	IF NOT FAULT THEN 
		oaksGVL.rOutdoorTempErrorValue0 := PV; // global utetemp som ställs till 0 vid givarfel.
		oaksGVL.rOutdoorTempErrorValue150 := PV;// global utetemp som ställs till 150 vid givarfel.
	ELSE
		oaksGVL.rOutdoorTempErrorValue0 := 0; // global utetemp som ställs till 0 vid givarfel.
		oaksGVL.rOutdoorTempErrorValue150 := 150;// global utetemp som ställs till 150 vid givarfel.
	END_IF
	oaksGVL.rOutdoorTempMean := PV1; // global medel utetemp
	
	oaksGVL.bOutdoorTempSensorError := FAULT; // globalt utegivarfel

METHOD PRIVATE mMean : BOOL // metod för att sköta uträkning av medelvärde
VAR_INPUT
END_VAR
	FB_BA_GetTime01(bEn :=TRUE);	
	stTime := FB_BA_GetTime01.stSysTi;

	IF stTime.wMinute <> wLastMinuteOfChange THEN
		fbMinuteTrig(CLK := TRUE);
	ELSE
		fbMinuteTrig(CLK := FALSE);
	END_IF
	//4320 minuter - 1 = 72 timmar.
	IF fbMinuteTrig.Q THEN
		FOR iCounter:= iAntalMinuterMedel - 1 TO 1 BY -1 DO
			rArrayMean72Hours[iCounter]:=rArrayMean72Hours[iCounter-1];
		END_FOR;
		rArrayMean72Hours[0] := PV;
		wLastMinuteOfChange := stTime.wMinute;
		IF PV6 < 4320 THEN // Räknas upp för att hålla koll på antal insamlade minuter
			PV6 := PV6 +1;
		END_IF
	END_IF 
	
	lrMeanInternal := 0;
	//4320 minuter - 1 = 72 timmar.
	iAntalMinuterForUtrakning := MIN(iAntalMinuterMedel,PV6); // Max begränsar antal minuter som används för beräkning beroende på hur många minuter som finns insamlade
	FOR iCounter:= iAntalMinuterForUtrakning TO 1 BY -1 DO
		lrMeanInternalTemp := lrMeanInternal;
		lrMeanInternal:=rArrayMean72Hours[iCounter-1] + lrMeanInternalTemp;
	END_FOR;
END_METHOD

//utetemp som behåller sitt senaste giltiga värde vid givarfel 
METHOD PROTECTED mPv : REAL
VAR_INPUT
	bKeepLastValidData : BOOL;
END_VAR



	IF M THEN
		mPv := OPM;
	ELSIF FB_BA_AI01Temperatur.bWireBreak AND NOT bKeepLastValidData THEN
		mPv := 150;
	ELSIF FB_BA_AI01Temperatur.bShortCircuit AND NOT bKeepLastValidData THEN
		mPv := -50;
	ELSE
		mPv := LREAL_TO_REAL(FB_BA_TiAvrg01Temperatur.lrOut) + rCal;
	END_IF
END_METHOD

END_FUNCTION_BLOCK

// oaksLibrary/Givare/fbVoltageLuxLightCon
// 0-10V block med inbyggda taggar för ljusintensitet (lux) med möjlighet att handställa PV-värde och inbyggt lux-villkor för utebelysning. 
//Larmar vid givarfel eller vid handställning.
FUNCTION_BLOCK fbVoltageLuxLightCon
VAR_INPUT
	rLuxScaleX1 : REAL; // Ändra om det är 2-10V exempelvis. Max är 0..32767 så 2-10V = 32767 * 0.2 = 6553
	rLuxScaleX2 : REAL := 32767;
	rLuxScaleMin : REAL := 0;
	rLuxScaleMax : REAL := 10000;
	nErrorConf :UINT;//0=ej givarfel vid scalemin/max, 1=givarefel vid scalemax, 2=givarefel vid scalemin och scalemax
END_VAR
VAR_OUTPUT
	{attribute 'OPC.UA.DA' := '1'}
	PV2 AT %M* : REAL;//Ljusintensitet~wp:[unit]lux[format]0[trendoptions]i:300
	{attribute 'OPC.UA.DA' := '1'}
	AL6 AT %M* : BOOL;//Givarfel luxmätning~wp:
	{attribute 'OPC.UA.DA' := '1'}
	PV8 AT %M* : STRING := '';  //Skalning lux-givare~wp:
	{attribute 'OPC.UA.DA' := '1'}
	V AT %M* : BOOL; //Belysningssvillkor utebel.~wp:[trendoptions]i:14400, t:1
END_VAR
VAR
	usiStateLux AT %I*: USINT;
	iDataInLux AT %I*: INT;
	usiCtrlLux AT %Q*: USINT;
	iDataOutLux AT %Q*: INT;
	FB_BA_AI01Lux : FB_BA_AI;
	FB_BA_TiAvrg01Lux : tc2_ba.FB_BA_TiAvrg;
	sTempLux : STRING;
	fbTON : TON ; 
	
	fbTonBelysningsvillkor : TON;
	fbTofBelysningsvillkor : TOF;
END_VAR
VAR_INPUT PERSISTENT 
	{attribute 'OPC.UA.DA' := '1'}
	SP2 AT %M* : REAL := 400;//Gränsvärde start utebelysning.~wp:[unit]lux[format]0
	{attribute 'OPC.UA.DA' := '1'}
	SP3 AT %M*: REAL := 30;//Till & frånslag tidsfördr.~wp:[unit]min[format]0
	rCal : REAL; // Kalibrering
	iLuxMedelvardeSekunder : UDINT := 180;
END_VAR

	sTempLux := CONCAT(REAL_TO_STRING(rLuxScaleMin),' - '); 
	PV8 := CONCAT(sTempLux,REAL_TO_STRING(rLuxScaleMax)); 
	FB_BA_AI01Lux(
	TI_usiState:= usiStateLux, 
	TI_iDataIn:= iDataInLux, 
	eTerminal:= 17, 
	eSensor:= 0, (* 0 = pt1000, *)
	bConfigurate:= , 
	rX01:=rLuxScaleX1 , 
	rX02:=rLuxScaleX2 , 
	rY01:= rLuxScaleMin, 
	rY02:= rLuxScaleMax, 
	rOffset:= , 
	rSmoothingFactor:= , 
	udiDecimalPlace:= , 
	bEnLimitCtrl:= , 
	rHighLimit:= , 
	rLowLimit:=, 
	udiDelayLimitCtrl_sec:= , 
	TO_usiCtrl=> usiCtrlLux, 
	TO_iDataOut=> iDataOutLux, 
	rVal=> , 
	bWireBreak=> , 
	bShortCircuit=> , 
	bHighLimit=> , 
	bLowLimit=> , 
	bErr=> , 
	sErrDescr=> );
	
	FB_BA_TiAvrg01Lux(
	bEn:= TRUE, 
	bEnAvrg := TRUE,
	lrIn:=REAL_TO_LREAL(FB_BA_AI01Lux.rVal), 
	udiIntval:=1, 
	udiNumOfElem:= iLuxMedelvardeSekunder, 
	lrOut=> );
	PV2 := LREAL_TO_REAL(FB_BA_TiAvrg01Lux.lrOut) +rCal;
	
	//Givarfel vid rangemin/max
	IF nErrorConf = 1 THEN 
		fbTON.IN := PV2 >= rLuxScaleMin - 1;
	ELSIF nErrorConf = 2 THEN 
		fbTON.IN := (PV2 >= rLuxScaleMin - 1) OR (PV2 <= rLuxScaleMax + 1);
	ELSE
		fbTON.IN := 0;
	END_IF
	
	fbTON(PT := T#5S);
	AL6 := FB_BA_AI01Lux.bWireBreak OR FB_BA_AI01Lux.bShortCircuit OR fbTON.Q;
	
	// Till och frånslagsfördröjning ute utebelysningsvillkor (V)
	fbTonBelysningsvillkor(IN:=PV2 < SP2, PT:=fRealToMinute(SP3) , Q=> , ET=> );
	fbTofBelysningsvillkor(IN:=fbTonBelysningsvillkor.Q , PT:=fRealToMinute(SP3) , Q=>V , ET=> );

END_FUNCTION_BLOCK

// oaksLibrary/Givare/fbVoltage
//Generellt analog-in block för 0-10V/4-20mA mfl. Funktionsblock har möjlighet att handställa PV-värde. Larmar vid givarfel eller vid handställning.
//Funktionsblock hanterar samtliga modultyper tex. KL3454/64. iBusTermType (17=0-10V, 21=4-20mA). Se typer E_BA_Terminal_KL.
FUNCTION_BLOCK fbVoltage
VAR_INPUT
	rScaleX1 : REAL; // Ändra om det är 2-10V exempelvis. Max är 0..32767 så 2-10V = 32767 * 0.2 = 6553
	rScaleX2 : REAL := 32767;
	rScaleMin : REAL;
	rScaleMax : REAL;

	iBusTermType : E_BA_TERMINAL_KL := 17; //Bus-terminal typ
	{attribute 'OPC.UA.DA' := '1'}
	M AT %M* : BOOL;//Handställning~wp:[trendoptions]i:14400, t:1
	
	nErrorConf :UINT;//0=ej givarfel vid scalemin/max, 1=givarefel vid scalemax, 2=givarefel vid scalemin och scalemax
END_VAR
VAR_OUTPUT
	rOutput : REAL;//Utgång knyts till tagg
	{attribute 'OPC.UA.DA' := '1'}
	FAULT AT %M* : BOOL;//Givarfel~wp:
	{attribute 'OPC.UA.DA' := '1'}
	AL8 AT %M* : BOOL; //Givare handställd~wp:[alarmoptions]p:3
	{attribute 'OPC.UA.DA' := '1'}
	PV8 AT %M* : STRING := '';  //Skalning givare~wp:
END_VAR
VAR
	usiState AT %I*: USINT;
	iDataIn AT %I*: INT;
	usiCtrl AT %Q*: USINT;
	iDataOut AT %Q*: INT;
	FB_BA_AI01 : FB_BA_AI;
	FB_BA_TiAvrg01 : tc2_ba.FB_BA_TiAvrg;
	sTemp : STRING;
	fbTON : TON;
END_VAR
VAR_INPUT PERSISTENT 
	rHandsetValue : REAL; //OPM värde
	rCal : REAL; //Kalibrering
	iMedelvardeSekunder : UDINT := 5;
END_VAR

	sTemp := CONCAT(REAL_TO_STRING(rScaleMin),' - '); 
	PV8 := CONCAT(sTemp,REAL_TO_STRING(rScaleMax)); 
	
	FB_BA_AI01(
	TI_usiState:= usiState, 
	TI_iDataIn:= iDataIn, 
	eTerminal:= iBusTermType, 
	eSensor:= 0, (* 0 = pt1000, *)
	bConfigurate:= , 
	rX01:=rScaleX1 , 
	rX02:=rScaleX2 , 
	rY01:= rScaleMin, 
	rY02:= rScaleMax, 
	rOffset:= , 
	rSmoothingFactor:= , 
	udiDecimalPlace:= , 
	bEnLimitCtrl:= , 
	rHighLimit:= , 
	rLowLimit:=, 
	udiDelayLimitCtrl_sec:= , 
	TO_usiCtrl=> usiCtrl, 
	TO_iDataOut=> iDataOut, 
	rVal=> , 
	bWireBreak=> , 
	bShortCircuit=> , 
	bHighLimit=> , 
	bLowLimit=> , 
	bErr=> , 
	sErrDescr=> );
	
	FB_BA_TiAvrg01(
	bEn:= TRUE, 
	bEnAvrg := TRUE,
	lrIn:=REAL_TO_LREAL(FB_BA_AI01.rVal), 
	udiIntval:=1, 
	udiNumOfElem:= iMedelvardeSekunder, 
	lrOut=> );
	
	
	AL8 := M;
	
	IF M THEN
		rOutput := rHandsetValue;
	ELSE 
		rOutput := LREAL_TO_REAL(FB_BA_TiAvrg01.lrOut) + rCal;
	END_IF
	
	//Givarfel vid rangemin/max
	IF nErrorConf = 1 THEN 
		fbTON.IN := rOutput >= rScaleMax - 1;
	ELSIF nErrorConf = 2 THEN 
		fbTON.IN := (rOutput >= rScaleMax - 1) OR (rOutput <= rScaleMin + 1);
	ELSE
		fbTON.IN := 0;
	END_IF
	
	fbTON(PT := T#5S);
	FAULT := FB_BA_AI01.bWireBreak OR FB_BA_AI01.bShortCircuit OR fbTON.Q;

END_FUNCTION_BLOCK

// oaksLibrary/Givare/fbVoltageBar
// 0-10V block med inbyggda taggar för tryck (kPa) med möjlighet att handställa PV-värde. Larmar vid givarfel eller vid handställning.
FUNCTION_BLOCK fbVoltageBar
VAR_INPUT
	rScaleX1 : REAL; // Ändra om det är 2-10V exempelvis. Max är 0..32767 så 2-10V = 32767 * 0.2 = 6553
	rScaleX2 : REAL := 32767;
	rScaleMin : REAL;
	rScaleMax : REAL;
	{attribute 'OPC.UA.DA' := '1'}
	M AT %M* : BOOL;//Handställning~wp:[trendoptions]i:14400, t:1
	nErrorConf :UINT;//0=ej givarfel vid scalemin/max, 1=givarefel vid scalemax, 2=givarefel vid scalemin och scalemax
END_VAR
VAR_OUTPUT
	{attribute 'OPC.UA.DA' := '1'}
	PV AT %M* : REAL;//Tryck~wp:[unit]Bar[format]0.0[trendoptions]i:300
	{attribute 'OPC.UA.DA' := '1'}
	FAULT AT %M* : BOOL;//Givarfel~wp:
	{attribute 'OPC.UA.DA' := '1'}
	AL8 AT %M* : BOOL; //Givare handställd~wp:[alarmoptions]p:3
	{attribute 'OPC.UA.DA' := '1'}
	PV8 AT %M* : STRING := '';  //Skalning givare~wp:
END_VAR
VAR
	fbAlarm2 : fbAlarm; // Larm handställning
	usiState AT %I*: USINT;
	iDataIn AT %I*: INT;
	usiCtrl AT %Q*: USINT;
	iDataOut AT %Q*: INT;
	FB_BA_AI01 : FB_BA_AI;
	FB_BA_TiAvrg01 : tc2_ba.FB_BA_TiAvrg;
	sTemp : STRING;
	fbTON : TON ; 
END_VAR
VAR_INPUT PERSISTENT
	{attribute 'OPC.UA.DA' := '1'}
	OPM AT %M* : REAL;//Värde handställning~wp:[unit]Bar[format]0.0
	rCal : REAL; // Kalibrering
	iMedelvardeSekunder : UDINT := 5;
END_VAR

	sTemp := CONCAT(REAL_TO_STRING(rScaleMin),' - '); 
	PV8 := CONCAT(sTemp,REAL_TO_STRING(rScaleMax)); 

	FB_BA_AI01(
	TI_usiState:= usiState, 
	TI_iDataIn:= iDataIn, 
	eTerminal:= 17, 
	eSensor:= 0, (* 0 = pt1000, *)
	bConfigurate:= , 
	rX01:=rScaleX1 , 
	rX02:=rScaleX2 , 
	rY01:= rScaleMin, 
	rY02:= rScaleMax, 
	rOffset:= , 
	rSmoothingFactor:= , 
	udiDecimalPlace:= , 
	bEnLimitCtrl:= , 
	rHighLimit:= , 
	rLowLimit:=, 
	udiDelayLimitCtrl_sec:= , 
	TO_usiCtrl=> usiCtrl, 
	TO_iDataOut=> iDataOut, 
	rVal=> , 
	bWireBreak=> , 
	bShortCircuit=> , 
	bHighLimit=> , 
	bLowLimit=> , 
	bErr=> , 
	sErrDescr=> );
	
	FB_BA_TiAvrg01(
	bEn:= TRUE, 
	bEnAvrg := TRUE,
	lrIn:=REAL_TO_LREAL(FB_BA_AI01.rVal), 
	udiIntval:=1, 
	udiNumOfElem:= iMedelvardeSekunder, 
	lrOut=> );
	
	
	//Handställningslarm
	fbAlarm2(bInput:=M , tAlarmDelay:= , bAutoReset:=TRUE , bAlarmOutput=>AL8 );
	
	IF M THEN
		PV := OPM;
	ELSE 
		PV := LREAL_TO_REAL(FB_BA_TiAvrg01.lrOut) +rCal;
	END_IF
	
	//Givarfel vid rangemin/max
	IF nErrorConf = 1 THEN 
		fbTON.IN := PV >= rScaleMax - 1;
	ELSIF nErrorConf = 2 THEN 
		fbTON.IN := (PV >= rScaleMax - 1) OR (PV <= rScaleMin + 1);
	ELSE
		fbTON.IN := 0;
	END_IF
	
	fbTON(PT := T#5S);
	FAULT := FB_BA_AI01.bWireBreak OR FB_BA_AI01.bShortCircuit OR fbTON.Q;

END_FUNCTION_BLOCK

// oaksLibrary/Givare/fbVoltageCo
// 0-10V block med inbyggda taggar för Kolmonoxid (ppm) med möjlighet att handställa PV-värde. Larmar vid givarfel eller vid handställning.
FUNCTION_BLOCK fbVoltageCo
VAR_INPUT
	rScaleX1 : REAL; // Ändra om det är 2-10V exempelvis. Max är 0..32767 så 2-10V = 32767 * 0.2 = 6553
	rScaleX2 : REAL := 32767;
	rScaleMin : REAL;
	rScaleMax : REAL;
	{attribute 'OPC.UA.DA' := '1'}
	M AT %M* : BOOL;//Handställning~wp:[trendoptions]i:14400, t:1
	nErrorConf :UINT;//0=ej givarfel vid scalemin/max, 1=givarefel vid scalemax, 2=givarefel vid scalemin och scalemax
END_VAR
VAR_OUTPUT
	{attribute 'OPC.UA.DA' := '1'}
	PV AT %M* : REAL;//Kolmonoxid~wp:[unit]ppm[format]0[trendoptions]i:300
	{attribute 'OPC.UA.DA' := '1'}
	FAULT AT %M* : BOOL;//Givarfel~wp:
	{attribute 'OPC.UA.DA' := '1'}
	AL8 AT %M* : BOOL; //Givare handställd~wp:[alarmoptions]p:3
	{attribute 'OPC.UA.DA' := '1'}
	PV8 AT %M* : STRING := '';  //Skalning givare~wp:
END_VAR
VAR
	fbAlarm2 : fbAlarm; // Larm handställning
	usiState AT %I*: USINT;
	iDataIn AT %I*: INT;
	usiCtrl AT %Q*: USINT;
	iDataOut AT %Q*: INT;
	FB_BA_AI01 : FB_BA_AI;
	FB_BA_TiAvrg01 : tc2_ba.FB_BA_TiAvrg;
	sTemp : STRING;
	fbTON : TON ; 
END_VAR
VAR_INPUT PERSISTENT 
	{attribute 'OPC.UA.DA' := '1'}
	OPM AT %M* : REAL;//Värde handställning~wp:[unit]ppm[format]0
	rCal : REAL; // Kalibrering
	iMedelvardeSekunder : UDINT := 5;
END_VAR

	sTemp := CONCAT(REAL_TO_STRING(rScaleMin),' - '); 
	PV8 := CONCAT(sTemp,REAL_TO_STRING(rScaleMax)); 

	FB_BA_AI01(
	TI_usiState:= usiState, 
	TI_iDataIn:= iDataIn, 
	eTerminal:= 17, 
	eSensor:= 0, (* 0 = pt1000, *)
	bConfigurate:= , 
	rX01:=rScaleX1 , 
	rX02:=rScaleX2 , 
	rY01:= rScaleMin, 
	rY02:= rScaleMax, 
	rOffset:= , 
	rSmoothingFactor:= , 
	udiDecimalPlace:= , 
	bEnLimitCtrl:= , 
	rHighLimit:= , 
	rLowLimit:=, 
	udiDelayLimitCtrl_sec:= , 
	TO_usiCtrl=> usiCtrl, 
	TO_iDataOut=> iDataOut, 
	rVal=> , 
	bWireBreak=> , 
	bShortCircuit=> , 
	bHighLimit=> , 
	bLowLimit=> , 
	bErr=> , 
	sErrDescr=> );
	
	FB_BA_TiAvrg01(
	bEn:= TRUE, 
	bEnAvrg := TRUE,
	lrIn:=REAL_TO_LREAL(FB_BA_AI01.rVal), 
	udiIntval:=1, 
	udiNumOfElem:= iMedelvardeSekunder, 
	lrOut=> );
	
	
	//Handställningslarm
	fbAlarm2(bInput:=M , tAlarmDelay:= , bAutoReset:=TRUE , bAlarmOutput=>AL8 );
	
	IF M THEN
		PV := OPM;
	ELSE 
		PV := LREAL_TO_REAL(FB_BA_TiAvrg01.lrOut) +rCal;
	END_IF
	
	//Givarfel vid rangemin/max
	IF nErrorConf = 1 THEN 
		fbTON.IN := PV >= rScaleMax - 1;
	ELSIF nErrorConf = 2 THEN 
		fbTON.IN := (PV >= rScaleMax - 1) OR (PV <= rScaleMin + 1);
	ELSE
		fbTON.IN := 0;
	END_IF
	
	fbTON(PT := T#5S);
	FAULT := FB_BA_AI01.bWireBreak OR FB_BA_AI01.bShortCircuit OR fbTON.Q;

END_FUNCTION_BLOCK

// oaksLibrary/Givare/fbVoltageCo2
// 0-10V block med inbyggda taggar för tryck (kPa) med möjlighet att handställa PV-värde. Larmar vid givarfel eller vid handställning.
FUNCTION_BLOCK fbVoltageCo2
VAR_INPUT
	rScaleX1 : REAL; // Ändra om det är 2-10V exempelvis. Max är 0..32767 så 2-10V = 32767 * 0.2 = 6553
	rScaleX2 : REAL := 32767;
	rScaleMin : REAL;
	rScaleMax : REAL;
	{attribute 'OPC.UA.DA' := '1'}
	M AT %M* : BOOL;//Handställning~wp:[trendoptions]i:14400, t:1
	nErrorConf :UINT;//0=ej givarfel vid scalemin/max, 1=givarefel vid scalemax, 2=givarefel vid scalemin och scalemax
END_VAR
VAR_OUTPUT
	{attribute 'OPC.UA.DA' := '1'}
	PV AT %M* : REAL;//Co2-halt~wp:[unit]ppm[format]0[trendoptions]i:300
	{attribute 'OPC.UA.DA' := '1'}
	FAULT AT %M* : BOOL;//Givarfel~wp:
	{attribute 'OPC.UA.DA' := '1'}
	AL8 AT %M* : BOOL; //Givare handställd~wp:[alarmoptions]p:3
	{attribute 'OPC.UA.DA' := '1'}
	PV8 AT %M* : STRING := '';  //Skalning givare~wp:
END_VAR
VAR
	fbAlarm2 : fbAlarm; // Larm handställning
	usiState AT %I*: USINT;
	iDataIn AT %I*: INT;
	usiCtrl AT %Q*: USINT;
	iDataOut AT %Q*: INT;
	FB_BA_AI01 : FB_BA_AI;
	FB_BA_TiAvrg01 : tc2_ba.FB_BA_TiAvrg;
	sTemp : STRING;
	fbTON : TON ; 
END_VAR
VAR_INPUT PERSISTENT
	{attribute 'OPC.UA.DA' := '1'}
	OPM AT %M* : REAL;//Värde handställning~wp:[unit]ppm[format]0
	rCal : REAL; // Kalibrering
	iMedelvardeSekunder : UDINT := 5;
END_VAR

	sTemp := CONCAT(REAL_TO_STRING(rScaleMin),' - '); 
	PV8 := CONCAT(sTemp,REAL_TO_STRING(rScaleMax)); 

	FB_BA_AI01(
	TI_usiState:= usiState, 
	TI_iDataIn:= iDataIn, 
	eTerminal:= 17, 
	eSensor:= 0, (* 0 = pt1000, *)
	bConfigurate:= , 
	rX01:=rScaleX1 , 
	rX02:=rScaleX2 , 
	rY01:= rScaleMin, 
	rY02:= rScaleMax, 
	rOffset:= , 
	rSmoothingFactor:= , 
	udiDecimalPlace:= , 
	bEnLimitCtrl:= , 
	rHighLimit:= , 
	rLowLimit:=, 
	udiDelayLimitCtrl_sec:= , 
	TO_usiCtrl=> usiCtrl, 
	TO_iDataOut=> iDataOut, 
	rVal=> , 
	bWireBreak=> , 
	bShortCircuit=> , 
	bHighLimit=> , 
	bLowLimit=> , 
	bErr=> , 
	sErrDescr=> );
	
	FB_BA_TiAvrg01(
	bEn:= TRUE, 
	bEnAvrg := TRUE,
	lrIn:=REAL_TO_LREAL(FB_BA_AI01.rVal), 
	udiIntval:=1, 
	udiNumOfElem:= iMedelvardeSekunder, 
	lrOut=> );
	
	
	//Handställningslarm
	fbAlarm2(bInput:=M , tAlarmDelay:= , bAutoReset:=TRUE , bAlarmOutput=>AL8 );
	
	IF M THEN
		PV := OPM;
	ELSE 
		PV := LREAL_TO_REAL(FB_BA_TiAvrg01.lrOut) +rCal;
	END_IF
	
	//Givarfel vid rangemin/max
	IF nErrorConf = 1 THEN 
		fbTON.IN := PV >= rScaleMax - 1;
	ELSIF nErrorConf = 2 THEN 
		fbTON.IN := (PV >= rScaleMax - 1) OR (PV <= rScaleMin + 1);
	ELSE
		fbTON.IN := 0;
	END_IF
	
	fbTON(PT := T#5S);
	FAULT := FB_BA_AI01.bWireBreak OR FB_BA_AI01.bShortCircuit OR fbTON.Q;

END_FUNCTION_BLOCK

// oaksLibrary/Givare/fbVoltagekPa
// 0-10V block med inbyggda taggar för tryck (kPa) med möjlighet att handställa PV-värde. Larmar vid givarfel eller vid handställning.
FUNCTION_BLOCK fbVoltagekPa
VAR_INPUT
	rScaleX1 : REAL; // Ändra om det är 2-10V exempelvis. Max är 0..32767 så 2-10V = 32767 * 0.2 = 6553
	rScaleX2 : REAL := 32767;
	rScaleMin : REAL;
	rScaleMax : REAL;
	{attribute 'OPC.UA.DA' := '1'}
	M AT %M* : BOOL;//Handställning~wp:[trendoptions]i:14400, t:1
	nErrorConf :UINT;//0=ej givarfel vid scalemin/max, 1=givarefel vid scalemax, 2=givarefel vid scalemin och scalemax
END_VAR
VAR_OUTPUT
	{attribute 'OPC.UA.DA' := '1'}
	PV AT %M* : REAL;//Tryck~wp:[unit]kPa[format]0[trendoptions]i:300
	{attribute 'OPC.UA.DA' := '1'}
	FAULT AT %M* : BOOL;//Givarfel~wp:
	{attribute 'OPC.UA.DA' := '1'}
	AL8 AT %M* : BOOL; //Givare handställd~wp:[alarmoptions]p:3
	{attribute 'OPC.UA.DA' := '1'}
	PV8 AT %M* : STRING := '';  //Skalning givare~wp:
END_VAR
VAR
	fbAlarm2 : fbAlarm; // Larm handställning
	usiState AT %I*: USINT;
	iDataIn AT %I*: INT;
	usiCtrl AT %Q*: USINT;
	iDataOut AT %Q*: INT;
	FB_BA_AI01 : FB_BA_AI;
	FB_BA_TiAvrg01 : tc2_ba.FB_BA_TiAvrg;
	sTemp : STRING;
	fbTON : TON ; 
END_VAR
VAR_INPUT PERSISTENT
	{attribute 'OPC.UA.DA' := '1'} 
	OPM AT %M* : REAL;//Värde handställning~wp:[unit]kPa[format]0
	rCal : REAL; // Kalibrering
	iMedelvardeSekunder : UDINT := 5;
END_VAR

	sTemp := CONCAT(REAL_TO_STRING(rScaleMin),' - '); 
	PV8 := CONCAT(sTemp,REAL_TO_STRING(rScaleMax)); 

	FB_BA_AI01(
	TI_usiState:= usiState, 
	TI_iDataIn:= iDataIn, 
	eTerminal:= 17, 
	eSensor:= 0, (* 0 = pt1000, *)
	bConfigurate:= , 
	rX01:=rScaleX1 , 
	rX02:=rScaleX2 , 
	rY01:= rScaleMin, 
	rY02:= rScaleMax, 
	rOffset:= , 
	rSmoothingFactor:= , 
	udiDecimalPlace:= , 
	bEnLimitCtrl:= , 
	rHighLimit:= , 
	rLowLimit:=, 
	udiDelayLimitCtrl_sec:= , 
	TO_usiCtrl=> usiCtrl, 
	TO_iDataOut=> iDataOut, 
	rVal=> , 
	bWireBreak=> , 
	bShortCircuit=> , 
	bHighLimit=> , 
	bLowLimit=> , 
	bErr=> , 
	sErrDescr=> );
	
	FB_BA_TiAvrg01(
	bEn:= TRUE, 
	bEnAvrg := TRUE,
	lrIn:=REAL_TO_LREAL(FB_BA_AI01.rVal), 
	udiIntval:=1, 
	udiNumOfElem:= iMedelvardeSekunder, 
	lrOut=> );
	
	
	//Handställningslarm
	fbAlarm2(bInput:=M , tAlarmDelay:= , bAutoReset:=TRUE , bAlarmOutput=>AL8 );
	
	IF M THEN
		PV := OPM;
	ELSE 
		PV := LREAL_TO_REAL(FB_BA_TiAvrg01.lrOut) +rCal;
	END_IF
	
	//Givarfel vid rangemin/max
	IF nErrorConf = 1 THEN 
		fbTON.IN := PV >= rScaleMax - 1;
	ELSIF nErrorConf = 2 THEN 
		fbTON.IN := (PV >= rScaleMax - 1) OR (PV <= rScaleMin + 1);
	ELSE
		fbTON.IN := 0;
	END_IF
	
	fbTON(PT := T#5S);
	FAULT := FB_BA_AI01.bWireBreak OR FB_BA_AI01.bShortCircuit OR fbTON.Q;

END_FUNCTION_BLOCK

// oaksLibrary/Givare/fbVoltageLs
//Oaks AB
//2022-03-11
//0-10V block med inbyggda taggar för flöde (L/s) med möjlighet att handställa PV-värde. Larmar vid givarfel eller vid handställning.
FUNCTION_BLOCK fbVoltageLs
VAR_INPUT
	rScaleX1 : REAL; // Ändra om det är 2-10V exempelvis. Max är 0..32767 så 2-10V = 32767 * 0.2 = 6553
	rScaleX2 : REAL := 32767;
	rScaleMin : REAL;
	rScaleMax : REAL;
	{attribute 'OPC.UA.DA' := '1'}
	M AT %M* : BOOL;//Handställning~wp:[trendoptions]i:14400, t:1
	nErrorConf :UINT;//0=ej givarfel vid scalemin/max, 1=givarefel vid scalemax, 2=givarefel vid scalemin och scalemax
END_VAR
VAR_OUTPUT
	{attribute 'OPC.UA.DA' := '1'}
	PV AT %M* : REAL;//Flöde~wp:[unit]l/s[format]0[trendoptions]i:300
	{attribute 'OPC.UA.DA' := '1'}
	FAULT AT %M* : BOOL;//Givarfel~wp:
	{attribute 'OPC.UA.DA' := '1'}
	AL8 AT %M* : BOOL; //Givare handställd~wp:[alarmoptions]p:3
	{attribute 'OPC.UA.DA' := '1'}
	PV8 AT %M* : STRING := '';  //Skalning givare~wp:
END_VAR
VAR
	fbAlarm2 : fbAlarm; //Larm handställning
	usiState AT %I*: USINT;
	iDataIn AT %I*: INT;
	usiCtrl AT %Q*: USINT;
	iDataOut AT %Q*: INT;
	FB_BA_AI01 : FB_BA_AI;
	FB_BA_TiAvrg01 : tc2_ba.FB_BA_TiAvrg;
	sTemp : STRING;
	fbTON : TON ; 
END_VAR
VAR_INPUT PERSISTENT 
	{attribute 'OPC.UA.DA' := '1'}
	OPM AT %M* : REAL;//Värde handställning~wp:[unit]l/s[format]0
	rCal : REAL; // Kalibrering
	iMedelvardeSekunder : UDINT := 5;
END_VAR

	sTemp := CONCAT(REAL_TO_STRING(rScaleMin),' - '); 
	PV8 := CONCAT(sTemp,REAL_TO_STRING(rScaleMax)); 

	FB_BA_AI01(
	TI_usiState:= usiState, 
	TI_iDataIn:= iDataIn, 
	eTerminal:= 17, 
	eSensor:= 0, (* 0 = pt1000, *)
	bConfigurate:= , 
	rX01:=rScaleX1 , 
	rX02:=rScaleX2 , 
	rY01:= rScaleMin, 
	rY02:= rScaleMax, 
	rOffset:= , 
	rSmoothingFactor:= , 
	udiDecimalPlace:= , 
	bEnLimitCtrl:= , 
	rHighLimit:= , 
	rLowLimit:=, 
	udiDelayLimitCtrl_sec:= , 
	TO_usiCtrl=> usiCtrl, 
	TO_iDataOut=> iDataOut, 
	rVal=> , 
	bWireBreak=> , 
	bShortCircuit=> , 
	bHighLimit=> , 
	bLowLimit=> , 
	bErr=> , 
	sErrDescr=> );
	
	FB_BA_TiAvrg01(
	bEn:= TRUE, 
	bEnAvrg := TRUE,
	lrIn:=REAL_TO_LREAL(FB_BA_AI01.rVal), 
	udiIntval:=1, 
	udiNumOfElem:= iMedelvardeSekunder, 
	lrOut=> );
	
	//Handställningslarm
	fbAlarm2(bInput:=M , tAlarmDelay:= , bAutoReset:=TRUE , bAlarmOutput=>AL8 );
	
	IF M THEN
		PV := OPM;
	ELSE 
		PV := LREAL_TO_REAL(FB_BA_TiAvrg01.lrOut) +rCal;
	END_IF
	
	//Givarfel vid rangemin/max
	IF nErrorConf = 1 THEN 
		fbTON.IN := PV >= rScaleMax - 1;
	ELSIF nErrorConf = 2 THEN 
		fbTON.IN := (PV >= rScaleMax - 1) OR (PV <= rScaleMin + 1);
	ELSE
		fbTON.IN := 0;
	END_IF
	
	fbTON(PT := T#5S);
	FAULT := FB_BA_AI01.bWireBreak OR FB_BA_AI01.bShortCircuit OR fbTON.Q;

END_FUNCTION_BLOCK

// oaksLibrary/Givare/fbVoltageLux
// 0-10V block med inbyggda taggar för ljusintensitet (lux) med möjlighet att handställa PV-värde. Larmar vid givarfel eller vid handställning.
FUNCTION_BLOCK fbVoltageLux
VAR_INPUT
	rScaleX1 : REAL; // Ändra om det är 2-10V exempelvis. Max är 0..32767 så 2-10V = 32767 * 0.2 = 6553
	rScaleX2 : REAL := 32767;
	rScaleMin : REAL;
	rScaleMax : REAL;
	{attribute 'OPC.UA.DA' := '1'}
	M AT %M* : BOOL;//Handställning luxgivare~wp:[trendoptions]i:14400, t:1
	nErrorConf :UINT;//0=ej givarfel vid scalemin/max, 1=givarefel vid scalemax, 2=givarefel vid scalemin och scalemax
END_VAR
VAR_OUTPUT
	{attribute 'OPC.UA.DA' := '1'}
	PV AT %M* : REAL;//Ljusintensitet~wp:[unit]lux[format]0[trendoptions]i:300
	{attribute 'OPC.UA.DA' := '1'}
	FAULT AT %M* : BOOL;//Givarfel~wp:
	{attribute 'OPC.UA.DA' := '1'}
	AL8 AT %M* : BOOL; //Givare handställd~wp:[alarmoptions]p:3
	{attribute 'OPC.UA.DA' := '1'}
	PV8 AT %M* : STRING := '';  //Skalning givare~wp:
END_VAR
VAR
	fbAlarm2 : fbAlarm; // Larm handställning
	usiState AT %I*: USINT;
	iDataIn AT %I*: INT;
	usiCtrl AT %Q*: USINT;
	iDataOut AT %Q*: INT;
	FB_BA_AI01 : FB_BA_AI;
	FB_BA_TiAvrg01 : tc2_ba.FB_BA_TiAvrg;
	sTemp : STRING;
	fbTON : TON ; 
END_VAR
VAR_INPUT PERSISTENT 
	{attribute 'OPC.UA.DA' := '1'}
	OPM AT %M* : REAL;//Värde handställning~wp:[unit]lux[format]0
	rCal : REAL; // Kalibrering
	iMedelvardeSekunder : UDINT := 5;
END_VAR

	sTemp := CONCAT(REAL_TO_STRING(rScaleMin),' - '); 
	PV8 := CONCAT(sTemp,REAL_TO_STRING(rScaleMax)); 
	FB_BA_AI01(
	TI_usiState:= usiState, 
	TI_iDataIn:= iDataIn, 
	eTerminal:= 17, 
	eSensor:= 0, (* 0 = pt1000, *)
	bConfigurate:= , 
	rX01:=rScaleX1 , 
	rX02:=rScaleX2 , 
	rY01:= rScaleMin, 
	rY02:= rScaleMax, 
	rOffset:= , 
	rSmoothingFactor:= , 
	udiDecimalPlace:= , 
	bEnLimitCtrl:= , 
	rHighLimit:= , 
	rLowLimit:=, 
	udiDelayLimitCtrl_sec:= , 
	TO_usiCtrl=> usiCtrl, 
	TO_iDataOut=> iDataOut, 
	rVal=> , 
	bWireBreak=> , 
	bShortCircuit=> , 
	bHighLimit=> , 
	bLowLimit=> , 
	bErr=> , 
	sErrDescr=> );
	
	FB_BA_TiAvrg01(
	bEn:= TRUE, 
	bEnAvrg := TRUE,
	lrIn:=REAL_TO_LREAL(FB_BA_AI01.rVal), 
	udiIntval:=1, 
	udiNumOfElem:= iMedelvardeSekunder, 
	lrOut=> );
	
	
	//Handställningslarm
	fbAlarm2(bInput:=M , tAlarmDelay:= , bAutoReset:=TRUE , bAlarmOutput=>AL8 );
	
	IF M THEN
		PV := OPM;
	ELSE 
		PV := LREAL_TO_REAL(FB_BA_TiAvrg01.lrOut) +rCal;
	END_IF
	
	//Givarfel vid rangemin/max
	IF nErrorConf = 1 THEN 
		fbTON.IN := PV >= rScaleMax - 1;
	ELSIF nErrorConf = 2 THEN 
		fbTON.IN := (PV >= rScaleMax - 1) OR (PV <= rScaleMin + 1);
	ELSE
		fbTON.IN := 0;
	END_IF
	
	fbTON(PT := T#5S);
	FAULT := FB_BA_AI01.bWireBreak OR FB_BA_AI01.bShortCircuit OR fbTON.Q;

END_FUNCTION_BLOCK

// oaksLibrary/Givare/fbVoltageNo2
// 0-10V block med inbyggda taggar för Kvävedioxid (ppm) med möjlighet att handställa PV-värde. Larmar vid givarfel eller vid handställning.
FUNCTION_BLOCK fbVoltageNo2
VAR_INPUT
	rScaleX1 : REAL; // Ändra om det är 2-10V exempelvis. Max är 0..32767 så 2-10V = 32767 * 0.2 = 6553
	rScaleX2 : REAL := 32767;
	rScaleMin : REAL;
	rScaleMax : REAL;
	{attribute 'OPC.UA.DA' := '1'}
	M AT %M* : BOOL;//Handställning~wp:[trendoptions]i:14400, t:1
	nErrorConf :UINT;//0=ej givarfel vid scalemin/max, 1=givarefel vid scalemax, 2=givarefel vid scalemin och scalemax
END_VAR
VAR_OUTPUT
	{attribute 'OPC.UA.DA' := '1'}
	PV AT %M* : REAL;//Kvävedioxid~wp:[unit]ppm[format]0.0[trendoptions]i:300
	{attribute 'OPC.UA.DA' := '1'}
	FAULT AT %M* : BOOL;//Givarfel~wp:
	{attribute 'OPC.UA.DA' := '1'}
	AL8 AT %M* : BOOL; //Givare handställd~wp:[alarmoptions]p:3
	{attribute 'OPC.UA.DA' := '1'}
	PV8 AT %M* : STRING := '';  //Skalning givare~wp:
END_VAR
VAR
	fbAlarm2 : fbAlarm; // Larm handställning
	usiState AT %I*: USINT;
	iDataIn AT %I*: INT;
	usiCtrl AT %Q*: USINT;
	iDataOut AT %Q*: INT;
	FB_BA_AI01 : FB_BA_AI;
	FB_BA_TiAvrg01 : tc2_ba.FB_BA_TiAvrg;
	sTemp : STRING;
	fbTON : TON ; 
END_VAR
VAR_INPUT PERSISTENT 
	{attribute 'OPC.UA.DA' := '1'}
	OPM AT %M* : REAL;//Värde handställning~wp:[unit]ppm[format]0.0
	rCal : REAL; // Kalibrering
	iMedelvardeSekunder : UDINT := 5;
END_VAR

	sTemp := CONCAT(REAL_TO_STRING(rScaleMin),' - '); 
	PV8 := CONCAT(sTemp,REAL_TO_STRING(rScaleMax)); 

	FB_BA_AI01(
	TI_usiState:= usiState, 
	TI_iDataIn:= iDataIn, 
	eTerminal:= 17, 
	eSensor:= 0, (* 0 = pt1000, *)
	bConfigurate:= , 
	rX01:=rScaleX1 , 
	rX02:=rScaleX2 , 
	rY01:= rScaleMin, 
	rY02:= rScaleMax, 
	rOffset:= , 
	rSmoothingFactor:= , 
	udiDecimalPlace:= , 
	bEnLimitCtrl:= , 
	rHighLimit:= , 
	rLowLimit:=, 
	udiDelayLimitCtrl_sec:= , 
	TO_usiCtrl=> usiCtrl, 
	TO_iDataOut=> iDataOut, 
	rVal=> , 
	bWireBreak=> , 
	bShortCircuit=> , 
	bHighLimit=> , 
	bLowLimit=> , 
	bErr=> , 
	sErrDescr=> );
	
	FB_BA_TiAvrg01(
	bEn:= TRUE, 
	bEnAvrg := TRUE,
	lrIn:=REAL_TO_LREAL(FB_BA_AI01.rVal), 
	udiIntval:=1, 
	udiNumOfElem:= iMedelvardeSekunder, 
	lrOut=> );
	
	
	//Handställningslarm
	fbAlarm2(bInput:=M , tAlarmDelay:= , bAutoReset:=TRUE , bAlarmOutput=>AL8 );
	
	IF M THEN
		PV := OPM;
	ELSE 
		PV := LREAL_TO_REAL(FB_BA_TiAvrg01.lrOut) +rCal;
	END_IF
	
	//Givarfel vid rangemin/max
	IF nErrorConf = 1 THEN 
		fbTON.IN := PV >= rScaleMax - 1;
	ELSIF nErrorConf = 2 THEN 
		fbTON.IN := (PV >= rScaleMax - 1) OR (PV <= rScaleMin + 1);
	ELSE
		fbTON.IN := 0;
	END_IF
	
	fbTON(PT := T#5S);
	FAULT := FB_BA_AI01.bWireBreak OR FB_BA_AI01.bShortCircuit OR fbTON.Q;

END_FUNCTION_BLOCK

// oaksLibrary/Givare/fbVoltagePa
// 0-10V block med inbyggda taggar för tryck (Pa) med möjlighet att handställa PV-värde. Larmar vid givarfel eller vid handställning.
FUNCTION_BLOCK fbVoltagePa
VAR_INPUT
	rScaleX1 : REAL; // Ändra om det är 2-10V exempelvis. Max är 0..32767 så 2-10V = 32767 * 0.2 = 6553
	rScaleX2 : REAL := 32767;
	rScaleMin : REAL;
	rScaleMax : REAL;
	{attribute 'OPC.UA.DA' := '1'}
	M AT %M* : BOOL;//Handställning~wp:[trendoptions]i:14400, t:1
	nErrorConf :UINT;//0=inget givarefel vid scalemin/max, 1=givarefel vid scalemax, 2=givarefel vid scalemin och scalemax
END_VAR
VAR_OUTPUT
	{attribute 'OPC.UA.DA' := '1'}
	PV AT %M* : REAL;//Tryck~wp:[unit]Pa[format]0[trendoptions]i:300
	{attribute 'OPC.UA.DA' := '1'}
	FAULT AT %M* : BOOL;//Givarfel~wp:
	{attribute 'OPC.UA.DA' := '1'}
	AL8 AT %M* : BOOL; //Givare handställd~wp:[alarmoptions]p:3
	{attribute 'OPC.UA.DA' := '1'}
	PV8 AT %M* : STRING := '';  //Skalning givare~wp:
END_VAR
VAR
	fbAlarm2 : fbAlarm; // Larm handställning
	usiState AT %I*: USINT;
	iDataIn AT %I*: INT;
	usiCtrl AT %Q*: USINT;
	iDataOut AT %Q*: INT;
	FB_BA_AI01 : FB_BA_AI;
	FB_BA_TiAvrg01 : tc2_ba.FB_BA_TiAvrg;
	sTemp : STRING;
	fbTON : TON ; 
END_VAR
VAR_INPUT PERSISTENT 
	{attribute 'OPC.UA.DA' := '1'}
	OPM AT %M* : REAL;//Värde handställning~wp:[unit]Pa[format]0
	rCal : REAL; // Kalibrering
	iMedelvardeSekunder : UDINT := 5;
END_VAR

	sTemp := CONCAT(REAL_TO_STRING(rScaleMin),' - '); 
	PV8 := CONCAT(sTemp,REAL_TO_STRING(rScaleMax)); 

	FB_BA_AI01(
	TI_usiState:= usiState, 
	TI_iDataIn:= iDataIn, 
	eTerminal:= 17, 
	eSensor:= 0, (* 0 = pt1000, *)
	bConfigurate:= , 
	rX01:=rScaleX1 , 
	rX02:=rScaleX2 , 
	rY01:= rScaleMin, 
	rY02:= rScaleMax, 
	rOffset:= , 
	rSmoothingFactor:= , 
	udiDecimalPlace:= , 
	bEnLimitCtrl:= , 
	rHighLimit:= , 
	rLowLimit:=, 
	udiDelayLimitCtrl_sec:= , 
	TO_usiCtrl=> usiCtrl, 
	TO_iDataOut=> iDataOut, 
	rVal=> , 
	bWireBreak=> , 
	bShortCircuit=> , 
	bHighLimit=> , 
	bLowLimit=> , 
	bErr=> , 
	sErrDescr=> );
	
	FB_BA_TiAvrg01(
	bEn:= TRUE, 
	bEnAvrg := TRUE,
	lrIn:=REAL_TO_LREAL(FB_BA_AI01.rVal), 
	udiIntval:=1, 
	udiNumOfElem:= iMedelvardeSekunder, 
	lrOut=> );
	
	
	//Handställningslarm
	fbAlarm2(bInput:=M , tAlarmDelay:= , bAutoReset:=TRUE , bAlarmOutput=>AL8 );
	
	IF M THEN
		PV := OPM;
	ELSE 
		PV := LREAL_TO_REAL(FB_BA_TiAvrg01.lrOut) +rCal;
	END_IF
	
	//Givarfel vid rangemin/max
	IF nErrorConf = 1 THEN 
		fbTON.IN := PV >= rScaleMax - 1;
	ELSIF nErrorConf = 2 THEN 
		fbTON.IN := (PV >= rScaleMax - 1) OR (PV <= rScaleMin + 1);
	ELSE
		fbTON.IN := 0;
	END_IF
	
	fbTON(PT := T#5S);
	FAULT := FB_BA_AI01.bWireBreak OR FB_BA_AI01.bShortCircuit OR fbTON.Q;

END_FUNCTION_BLOCK

// oaksLibrary/Givare/fbVoltagePaFlowLs
// Extendat fbVoltagePa med inbyggd tagg för uträknat flöde. Knyt ditt uträknade värde in på PV1
FUNCTION_BLOCK fbVoltagePaFlowLs EXTENDS fbVoltagePa
VAR_INPUT
	{attribute 'OPC.UA.DA' := '1'}
	PV1 AT %M* : REAL;//Uträknat flöde~wp:[unit]l/s[format]0[trendoptions]i:300
END_VAR
VAR_OUTPUT
END_VAR
VAR
END_VAR

SUPER^();

END_FUNCTION_BLOCK

// oaksLibrary/Givare/fbVoltageRh
// 0-10V block med inbyggda taggar för temperatur (rH%) med möjlighet att handställa PV-värde. Larmar vid givarfel eller vid handställning.
FUNCTION_BLOCK fbVoltageRh
VAR_INPUT
	rScaleX1 : REAL; // Ändra om det är 2-10V exempelvis. Max är 0..32767 så 2-10V = 32767 * 0.2 = 6553
	rScaleX2 : REAL := 32767;
	rScaleMin : REAL;
	rScaleMax : REAL;
	{attribute 'OPC.UA.DA' := '1'}
	M AT %M* : BOOL;//Handställning~wp:[trendoptions]i:14400, t:1
	nErrorConf :UINT;//0=ej givarfel vid scalemin/max, 1=givarefel vid scalemax, 2=givarefel vid scalemin och scalemax
END_VAR
VAR_OUTPUT
	{attribute 'OPC.UA.DA' := '1'}
	PV AT %M* : REAL;//Fukthalt~wp:[unit]rH%[format]0[trendoptions]i:300
	{attribute 'OPC.UA.DA' := '1'}
	FAULT AT %M* : BOOL;//Givarfel~wp:
	{attribute 'OPC.UA.DA' := '1'}
	AL8 AT %M* : BOOL; //Givare handställd~wp:[alarmoptions]p:3
	{attribute 'OPC.UA.DA' := '1'}
	PV8 AT %M* : STRING := '';  //Skalning givare~wp:
END_VAR
VAR
	fbAlarm2 : fbAlarm; // Larm handställning
	usiState AT %I*: USINT;
	iDataIn AT %I*: INT;
	usiCtrl AT %Q*: USINT;
	iDataOut AT %Q*: INT;
	FB_BA_AI01 : FB_BA_AI;
	FB_BA_TiAvrg01 : tc2_ba.FB_BA_TiAvrg;
	sTemp : STRING;
	fbTON : TON ; 
END_VAR
VAR_INPUT PERSISTENT
	{attribute 'OPC.UA.DA' := '1'}
	OPM AT %M* : REAL;//Värde handställning~wp:[unit]rH%[format]0
	rCal : REAL; // Kalibrering
	iMedelvardeSekunder : UDINT := 5;
END_VAR

sTemp := CONCAT(REAL_TO_STRING(rScaleMin),' - '); 
	PV8 := CONCAT(sTemp,REAL_TO_STRING(rScaleMax)); 

	FB_BA_AI01(
	TI_usiState:= usiState, 
	TI_iDataIn:= iDataIn, 
	eTerminal:= 17, 
	eSensor:= 0, (* 0 = pt1000, *)
	bConfigurate:= , 
	rX01:=rScaleX1 , 
	rX02:=rScaleX2 ,  
	rY01:= rScaleMin, 
	rY02:= rScaleMax, 
	rOffset:= , 
	rSmoothingFactor:= , 
	udiDecimalPlace:= , 
	bEnLimitCtrl:= , 
	rHighLimit:= , 
	rLowLimit:=, 
	udiDelayLimitCtrl_sec:= , 
	TO_usiCtrl=> usiCtrl, 
	TO_iDataOut=> iDataOut, 
	rVal=> , 
	bWireBreak=> , 
	bShortCircuit=> , 
	bHighLimit=> , 
	bLowLimit=> , 
	bErr=> , 
	sErrDescr=> );
	
	FB_BA_TiAvrg01(
	bEn:= TRUE, 
	bEnAvrg := TRUE,
	lrIn:=REAL_TO_LREAL(FB_BA_AI01.rVal), 
	udiIntval:=1, 
	udiNumOfElem:= iMedelvardeSekunder, 
	lrOut=> );
	
	
	//Handställningslarm
	fbAlarm2(bInput:=M , tAlarmDelay:= , bAutoReset:=TRUE , bAlarmOutput=>AL8 );
	
	IF M THEN
		PV := OPM;
	ELSE 
		PV := LREAL_TO_REAL(FB_BA_TiAvrg01.lrOut) +rCal;
	END_IF
	
	//Givarfel vid rangemin/max
	IF nErrorConf = 1 THEN 
		fbTON.IN := PV >= rScaleMax - 1;
	ELSIF nErrorConf = 2 THEN 
		fbTON.IN := (PV >= rScaleMax - 1) OR (PV <= rScaleMin + 1);
	ELSE
		fbTON.IN := 0;
	END_IF
	
	fbTON(PT := T#5S);
	FAULT := FB_BA_AI01.bWireBreak OR FB_BA_AI01.bShortCircuit OR fbTON.Q;

END_FUNCTION_BLOCK

// oaksLibrary/Givare/fbVoltageTemp
// 0-10V block med inbyggda taggar för temperatur (°C) med möjlighet att handställa PV-värde. Larmar vid givarfel eller vid handställning.
FUNCTION_BLOCK fbVoltageTemp
VAR_INPUT
	rScaleX1 : REAL; // Ändra om det är 2-10V exempelvis. Max är 0..32767 så 2-10V = 32767 * 0.2 = 6553
	rScaleX2 : REAL := 32767;
	rScaleMin : REAL;
	rScaleMax : REAL;
	{attribute 'OPC.UA.DA' := '1'}
	M AT %M* : BOOL;//Handställning~wp:[trendoptions]i:14400, t:1
	nErrorConf :UINT;//0=ej givarfel vid scalemin/max, 1=givarefel vid scalemax, 2=givarefel vid scalemin och scalemax
END_VAR
VAR_OUTPUT
	{attribute 'OPC.UA.DA' := '1'}
	PV AT %M* : REAL;//Temperatur~wp:[unit]°C[format]0.0[trendoptions]i:300
	{attribute 'OPC.UA.DA' := '1'}
	FAULT AT %M* : BOOL;//Givarfel~wp:
	{attribute 'OPC.UA.DA' := '1'}
	AL8 AT %M* : BOOL; //Givare handställd~wp:[alarmoptions]p:3
	{attribute 'OPC.UA.DA' := '1'}
	PV8 AT %M* : STRING := '';  //Skalning givare~wp:
END_VAR
VAR
	fbAlarm2 : fbAlarm; // Larm handställning
	usiState AT %I*: USINT;
	iDataIn AT %I*: INT;
	usiCtrl AT %Q*: USINT;
	iDataOut AT %Q*: INT;
	FB_BA_AI01 : FB_BA_AI;
	FB_BA_TiAvrg01 : tc2_ba.FB_BA_TiAvrg;
	sTemp : STRING;
	fbTON : TON ; 
END_VAR
VAR_INPUT PERSISTENT 
	{attribute 'OPC.UA.DA' := '1'}
	OPM AT %M* : REAL;//Värde handställning~wp:[unit]°C[format]0.0
	rCal : REAL; // Kalibrering
	iMedelvardeSekunder : UDINT := 5;
END_VAR

	sTemp := CONCAT(REAL_TO_STRING(rScaleMin),' - '); 
	PV8 := CONCAT(sTemp,REAL_TO_STRING(rScaleMax)); 

	FB_BA_AI01(
	TI_usiState:= usiState, 
	TI_iDataIn:= iDataIn, 
	eTerminal:= 17, 
	eSensor:= 0, (* 0 = pt1000, *)
	bConfigurate:= , 
	rX01:=rScaleX1 , 
	rX02:=rScaleX2 , 
	rY01:= rScaleMin, 
	rY02:= rScaleMax, 
	rOffset:= , 
	rSmoothingFactor:= , 
	udiDecimalPlace:= , 
	bEnLimitCtrl:= , 
	rHighLimit:= , 
	rLowLimit:=, 
	udiDelayLimitCtrl_sec:= , 
	TO_usiCtrl=> usiCtrl, 
	TO_iDataOut=> iDataOut, 
	rVal=> , 
	bWireBreak=> , 
	bShortCircuit=> , 
	bHighLimit=> , 
	bLowLimit=> , 
	bErr=> , 
	sErrDescr=> );
	
	FB_BA_TiAvrg01(
	bEn:= TRUE, 
	bEnAvrg := TRUE,
	lrIn:=REAL_TO_LREAL(FB_BA_AI01.rVal), 
	udiIntval:=1, 
	udiNumOfElem:= iMedelvardeSekunder, 
	lrOut=> );
	
	
	//Handställningslarm
	fbAlarm2(bInput:=M , tAlarmDelay:= , bAutoReset:=TRUE , bAlarmOutput=>AL8 );
	
	IF M THEN
		PV := OPM;
	ELSE 
		PV := LREAL_TO_REAL(FB_BA_TiAvrg01.lrOut) +rCal;
	END_IF
	
	//Givarfel vid rangemin/max
	IF nErrorConf = 1 THEN 
		fbTON.IN := PV >= rScaleMax - 1;
	ELSIF nErrorConf = 2 THEN 
		fbTON.IN := (PV >= rScaleMax - 1) OR (PV <= rScaleMin + 1);
	ELSE
		fbTON.IN := 0;
	END_IF
	
	fbTON(PT := T#5S);
	FAULT := FB_BA_AI01.bWireBreak OR FB_BA_AI01.bShortCircuit OR fbTON.Q;

END_FUNCTION_BLOCK

// oaksLibrary/Givare/fbVoltageTempCo2
// 0-10V block med inbyggda taggar för temperatur (°C) och CO2 (ppm) med möjlighet att handställa PV-värde. Larmar vid givarfel eller vid handställning.
FUNCTION_BLOCK fbVoltageTempCo2
VAR_INPUT
	rScaleX1Temperature : REAL; // Ändra om det är 2-10V exempelvis. Max är 0..32767 så 2-10V = 32767 * 0.2 = 6553
	rScaleX2Temperature : REAL := 32767;
	rScaleMinTemperature : REAL:=0;
	rScaleMaxTemperature : REAL:=50;
	
	rScaleX1Co2 : REAL; // Ändra om det är 2-10V exempelvis. Max är 0..32767 så 2-10V = 32767 * 0.2 = 6553
	rScaleX2Co2 : REAL := 32767;
	rScaleMinCo2 : REAL:=0;
	rScaleMaxCo2 : REAL:=2000;
	
	nErrorConfTemp :UINT;//0=inget givarefel 1=givarefel vid Scalemax 2=givarefel vid Scalemin och Scalemax
	nErrorConfCO2 :UINT;//0=inget givarefel 1=givarefel vid Scalemax 2=givarefel vid Scalemin och Scalemax
END_VAR
VAR_OUTPUT
	
	PV AT %M* : REAL;//Temperatur~wp:[unit]°C[format]0.0[trendoptions]i:300
	{attribute 'OPC.UA.DA' := '1'}
	PV1 AT %M* : REAL;//Co2-halt~wp:[unit]ppm[format]0[trendoptions]i:300
	{attribute 'OPC.UA.DA' := '1'}
	FAULT AT %M* : BOOL;//Givarfel temperatur~wp:
	{attribute 'OPC.UA.DA' := '1'}	
	AL8 AT %M* : BOOL;//Givarfel Co2~wp:
	{attribute 'OPC.UA.DA' := '1'}
	PV8 AT %M* : STRING := '';  //Skalning givare~wp:
END_VAR
VAR
	usiStateTemperature AT %I*: USINT;
	iDataInTemperature AT %I*: INT;
	usiCtrlTemperature AT %Q*: USINT;
	iDataOutTemperature AT %Q*: INT;
	FB_BA_AI_Temperature : FB_BA_AI;
	FB_BA_TiAvrgTemperature : tc2_ba.FB_BA_TiAvrg;
	
	usiStateCo2 AT %I*: USINT;
	iDataInCo2 AT %I*: INT;
	usiCtrlCo2 AT %Q*: USINT;
	iDataOutCo2 AT %Q*: INT;
	FB_BA_AI_Co2 : FB_BA_AI;
	FB_BA_TiAvrgCo2 : tc2_ba.FB_BA_TiAvrg;
	sTemp : STRING;
	fbTON1, fbTON2 : TON ;
END_VAR
VAR_INPUT PERSISTENT 
	rCalTemperature : REAL; // Kalibrering
	rCalCo2 : REAL; // Kalibrering
	iMedelvardeSekunder : UDINT := 5;
END_VAR

	

	sTemp := 'Temperatur: ';
	sTemp := CONCAT(CONCAT('Temperatur: ',REAL_TO_STRING(rScaleMinTemperature)),' - '); 
	sTemp := CONCAT(sTemp,REAL_TO_STRING(rScaleMaxTemperature)); 
	sTemp := CONCAT(sTemp,' , CO2: '); 
	sTemp := CONCAT(sTemp,REAL_TO_STRING(rScaleMinCo2)); 
	sTemp := CONCAT(sTemp, ' - ');  
	PV8 := CONCAT(sTemp,REAL_TO_STRING(rScaleMaxCo2));
(*************************** Temperatur *********************)	
	FB_BA_AI_Temperature(
	TI_usiState:= usiStateTemperature, 
	TI_iDataIn:= iDataInTemperature, 
	eTerminal:= 17, 
	eSensor:= 0, (* 0 = pt1000, *)
	bConfigurate:= , 
	rX01:=rScaleX1Temperature , 
	rX02:= rScaleX2Temperature, 
	rY01:= rScaleMinTemperature, 
	rY02:= rScaleMaxTemperature, 
	rOffset:= , 
	rSmoothingFactor:= , 
	udiDecimalPlace:= , 
	bEnLimitCtrl:= , 
	rHighLimit:= , 
	rLowLimit:=, 
	udiDelayLimitCtrl_sec:= , 
	TO_usiCtrl=> usiCtrlTemperature, 
	TO_iDataOut=> iDataOutTemperature, 
	rVal=> , 
	bWireBreak=> , 
	bShortCircuit=> , 
	bHighLimit=> , 
	bLowLimit=> , 
	bErr=> , 
	sErrDescr=> );
	
	FB_BA_TiAvrgTemperature(
	bEn:= TRUE, 
	bEnAvrg := TRUE,
	lrIn:=REAL_TO_LREAL(FB_BA_AI_Temperature.rVal), 
	udiIntval:=1, 
	udiNumOfElem:= iMedelvardeSekunder, 
	lrOut=> );
	
	PV := LREAL_TO_REAL(FB_BA_TiAvrgTemperature.lrOut) +rCalTemperature;
	
	//Givarfel vid rangemin/max
	IF nErrorConfTemp = 1 THEN 
		fbTON1.IN := PV >= rScaleMaxTemperature - 1;
	ELSIF nErrorConfTemp = 2 THEN 
		fbTON1.IN := (PV >= rScaleMaxTemperature - 1) OR (PV <= rScaleMinTemperature + 1);
	ELSE
		fbTON1.IN := 0;
	END_IF
	
	fbTON1(PT := T#5S); 
	
	FAULT := FB_BA_AI_Temperature.bWireBreak OR FB_BA_AI_Temperature.bShortCircuit OR fbTON1.Q;
(*************************** CO2 *********************)	
	FB_BA_AI_Co2(
	TI_usiState:= usiStateCo2, 
	TI_iDataIn:= iDataInCo2, 
	eTerminal:= 17, 
	eSensor:= 0, (* 0 = pt1000, *)
	bConfigurate:= , 
	rX01:= rScaleX1Co2, 
	rX02:= rScaleX2Co2, 
	rY01:= rScaleMinCo2, 
	rY02:= rScaleMaxCo2, 
	rOffset:= , 
	rSmoothingFactor:= , 
	udiDecimalPlace:= , 
	bEnLimitCtrl:= , 
	rHighLimit:= , 
	rLowLimit:=, 
	udiDelayLimitCtrl_sec:= , 
	TO_usiCtrl=> usiCtrlCo2, 
	TO_iDataOut=> iDataOutCo2, 
	rVal=> , 
	bWireBreak=> , 
	bShortCircuit=> , 
	bHighLimit=> , 
	bLowLimit=> , 
	bErr=> , 
	sErrDescr=> );
	
	FB_BA_TiAvrgCo2(
	bEn:= TRUE, 
	bEnAvrg := TRUE,
	lrIn:=REAL_TO_LREAL(FB_BA_AI_Co2.rVal), 
	udiIntval:=1, 
	udiNumOfElem:= iMedelvardeSekunder, 
	lrOut=> );
	
	PV1 := LREAL_TO_REAL(FB_BA_TiAvrgCo2.lrOut) +rCalCo2;
	
	//Givarfel vid rangemin/max
	IF nErrorConfCO2 = 1 THEN 
		fbTON2.IN := PV >= rScaleMaxCo2 - 1;
	ELSIF nErrorConfCO2 = 2 THEN 
		fbTON2.IN := (PV >= rScaleMaxCo2 - 1) OR (PV <= rScaleMinCo2 + 1);
	ELSE
		fbTON2.IN := 0;
	END_IF
	
	fbTON2(PT := T#5S);
	
	AL8 := FB_BA_AI_Co2.bWireBreak OR FB_BA_AI_Co2.bShortCircuit OR fbTON2.Q;

END_FUNCTION_BLOCK

// oaksLibrary/Givare/fbVoltageTempRh
// 0-10V block med inbyggda taggar för temperatur (°C) och rH (rH%) med möjlighet att handställa PV-värde. Larmar vid givarfel eller vid handställning.
FUNCTION_BLOCK fbVoltageTempRh
VAR_INPUT
	rScaleX1Temperature : REAL; // Ändra om det är 2-10V exempelvis. Max är 0..32767 så 2-10V = 32767 * 0.2 = 6553
	rScaleX2Temperature : REAL := 32767;
	rScaleMinTemperature : REAL:=0;
	rScaleMaxTemperature : REAL:=50;
	
	rScaleX1rH : REAL; // Ändra om det är 2-10V exempelvis. Max är 0..32767 så 2-10V = 32767 * 0.2 = 6553
	rScaleX2rH : REAL := 32767;
	rScaleMinrH : REAL:=0;
	rScaleMaxrH : REAL:=100;
	
	nErrorConfTemp :UINT;//0=inget givarefel 1=givarefel vid Scalemax 2=givarefel vid Scalemin och Scalemax
	nErrorConfrH :UINT;//0=inget givarefel 1=givarefel vid Scalemax 2=givarefel vid Scalemin och Scalemax

END_VAR
VAR_OUTPUT
	{attribute 'OPC.UA.DA' := '1'}
	PV AT %M* : REAL;//Temperatur~wp:[unit]°C[format]0.0[trendoptions]i:300
	{attribute 'OPC.UA.DA' := '1'}
	PV1 AT %M* : REAL;//rH-halt~wp:[unit]rH%[format]0[trendoptions]i:300
	{attribute 'OPC.UA.DA' := '1'}
	FAULT AT %M* : BOOL;//Givarfel temperatur~wp:
	{attribute 'OPC.UA.DA' := '1'}
	AL8 AT %M* : BOOL;//Givarfel rH~wp:
	{attribute 'OPC.UA.DA' := '1'}
	PV8 AT %M* : STRING := '';  //Skalning givare~wp:
END_VAR
VAR
	fbAlarm2 : fbAlarm; // Larm handställning
	usiStateTemperature AT %I*: USINT;
	iDataInTemperature AT %I*: INT;
	usiCtrlTemperature AT %Q*: USINT;
	iDataOutTemperature AT %Q*: INT;
	FB_BA_AI_Temperature : FB_BA_AI;
	FB_BA_TiAvrgTemperature : tc2_ba.FB_BA_TiAvrg;
	
	usiStaterH AT %I*: USINT;
	iDataInrH AT %I*: INT;
	usiCtrlrH AT %Q*: USINT;
	iDataOutrH AT %Q*: INT;
	FB_BA_AI_rH : FB_BA_AI;
	FB_BA_TiAvrgrH : tc2_ba.FB_BA_TiAvrg;
	sTemp : STRING;
	fbTON1, fbTON2 : TON ;
END_VAR
VAR_INPUT PERSISTENT 
	rCalTemperature : REAL; // Kalibrering
	rCalrH : REAL; // Kalibrering
	iMedelvardeSekunder : UDINT := 5;
END_VAR

	

	sTemp := 'Temperatur: ';
	sTemp := CONCAT(CONCAT('Temperatur: ',REAL_TO_STRING(rScaleMinTemperature)),' - '); 
	sTemp := CONCAT(sTemp,REAL_TO_STRING(rScaleMaxTemperature)); 
	sTemp := CONCAT(sTemp,' , rH%: '); 
	sTemp := CONCAT(sTemp,REAL_TO_STRING(rScaleMinrH)); 
	sTemp := CONCAT(sTemp, ' - ');  
	PV8 := CONCAT(sTemp,REAL_TO_STRING(rScaleMaxrH));
(*************************** Temperatur *********************)	
	FB_BA_AI_Temperature(
	TI_usiState:= usiStateTemperature, 
	TI_iDataIn:= iDataInTemperature, 
	eTerminal:= 17, 
	eSensor:= 0, (* 0 = pt1000, *)
	bConfigurate:= , 
	rX01:=rScaleX1Temperature , 
	rX02:= rScaleX2Temperature, 
	rY01:= rScaleMinTemperature, 
	rY02:= rScaleMaxTemperature, 
	rOffset:= , 
	rSmoothingFactor:= , 
	udiDecimalPlace:= , 
	bEnLimitCtrl:= , 
	rHighLimit:= , 
	rLowLimit:=, 
	udiDelayLimitCtrl_sec:= , 
	TO_usiCtrl=> usiCtrlTemperature, 
	TO_iDataOut=> iDataOutTemperature, 
	rVal=> , 
	bWireBreak=> , 
	bShortCircuit=> , 
	bHighLimit=> , 
	bLowLimit=> , 
	bErr=> , 
	sErrDescr=> );
	
	FB_BA_TiAvrgTemperature(
	bEn:= TRUE, 
	bEnAvrg := TRUE,
	lrIn:=REAL_TO_LREAL(FB_BA_AI_Temperature.rVal), 
	udiIntval:=1, 
	udiNumOfElem:= iMedelvardeSekunder, 
	lrOut=> );
	
	PV := LREAL_TO_REAL(FB_BA_TiAvrgTemperature.lrOut) +rCalTemperature;
	
	//Givarfel vid rangemin/max
	IF nErrorConfTemp = 1 THEN 
		fbTON1.IN := PV >= rScaleMaxTemperature - 1;
	ELSIF nErrorConfTemp = 2 THEN 
		fbTON1.IN := (PV >= rScaleMaxTemperature - 1) OR (PV <= rScaleMinTemperature + 1);
	ELSE
		fbTON1.IN := 0;
	END_IF
	
	fbTON1(PT := T#5S); 
	
	FAULT := FB_BA_AI_Temperature.bWireBreak OR FB_BA_AI_Temperature.bShortCircuit OR fbTON1.Q;
(*************************** rH *********************)	
	FB_BA_AI_rH(
	TI_usiState:= usiStaterH, 
	TI_iDataIn:= iDataInrH, 
	eTerminal:= 17, 
	eSensor:= 0, (* 0 = pt1000, *)
	bConfigurate:= , 
	rX01:= rScaleX1rH, 
	rX02:= rScaleX2rH, 
	rY01:= rScaleMinrH, 
	rY02:= rScaleMaxrH, 
	rOffset:= , 
	rSmoothingFactor:= , 
	udiDecimalPlace:= , 
	bEnLimitCtrl:= , 
	rHighLimit:= , 
	rLowLimit:=, 
	udiDelayLimitCtrl_sec:= , 
	TO_usiCtrl=> usiCtrlrH, 
	TO_iDataOut=> iDataOutrH, 
	rVal=> , 
	bWireBreak=> , 
	bShortCircuit=> , 
	bHighLimit=> , 
	bLowLimit=> , 
	bErr=> , 
	sErrDescr=> );
	
	FB_BA_TiAvrgrH(
	bEn:= TRUE, 
	bEnAvrg := TRUE,
	lrIn:=REAL_TO_LREAL(FB_BA_AI_rH.rVal), 
	udiIntval:=1, 
	udiNumOfElem:= iMedelvardeSekunder, 
	lrOut=> );
	
	PV1 := LREAL_TO_REAL(FB_BA_TiAvrgrH.lrOut) +rCalrH;
	
	//Givarfel vid rangemin/max
	IF nErrorConfRh = 1 THEN 
		fbTON2.IN := PV >= rScaleMaxrH - 1;
	ELSIF nErrorConfRh = 2 THEN 
		fbTON2.IN := (PV >= rScaleMaxrH - 1) OR (PV <= rScaleMinrH + 1);
	ELSE
		fbTON2.IN := 0;
	END_IF
	
	fbTON2(PT := T#5S);
	
	AL8 := FB_BA_AI_rH.bWireBreak OR FB_BA_AI_rH.bShortCircuit OR fbTON2.Q;

END_FUNCTION_BLOCK

// oaksLibrary/Hämta värde från Webport/fbOutDoorTempMeanFromScada
//Block för att läsa in utetemperatur från Webport. Larm utgår ifall värdet inte uppdateras på 48 timmar (inställningsbart).
(*
Skriv till PV i detta blocket i ett loopande script för uppdateringsvall på 10 sekunder enligt nedan.

tags["TAGG_ATT_HÄMTA_FRÅN_PV"].ReadValue(Moldeo.WebPortCommon.ReadTypes.PRIORITY); 
var copy = tags["TAGG_ATT_HÄMTA_FRÅN_PV"].Value; 
tags["DETTA_BLOCKETS_TAGG_PV"].WriteValue(copy, true); // Exempelvis AS02_GT31_PV

*)
FUNCTION_BLOCK fbOutDoorTempMeanFromScada
VAR_OUTPUT
	{attribute 'OPC.UA.DA' := '1'}
	PV AT %M* : REAL;//Temperatur~wp:[unit]°C[format]0.0[trendoptions]i:300
	{attribute 'OPC.UA.DA' := '1'}
	FAULT AT %M* : BOOL;//Kommunikationsfel hämtning av utetemperatur från webport~wp:
	{attribute 'OPC.UA.DA' := '1'}
	PV1 AT %M*  : REAL; //Medeltemperatur~wp:[unit]°C[format]0.0[trendoptions]i:300
END_VAR
VAR
	fbDifferenceCheckTemp: fbDifferenceCheck;
	fbAlarmTemp : fbAlarm;	

	bResetMeanTemp : BOOL; //Sätt denna till TRUE för återställning av medelvärdesberäkning.
	lrMeanInternal : LREAL;
	lrMeanInternalTemp : LREAL;
	fbPLC_SystemTime: Tc3_BA.FB_BA_GetTime;
	stTime		: tc2_ba.TIMESTRUCT;

	FB_BA_GetTime01 : tc2_ba.FB_BA_GetTime; 
	FB_BA_ExtTiSt01 : tc2_ba.FB_BA_ExtTiSt;	

	
	
	wMinute : WORD;
	fbMinuteTrig : R_TRIG;
	//iTemp : INT;
	iCounter : UINT := 4319;
	
	iAntalMinuterMedel : UINT;
	iAntalMinuterForUtrakning : UINT; //Maxbegränsar antal minuter som används för beräkning beroende på hur många minuter som finns insamlade
END_VAR
VAR PERSISTENT
	wLastMinuteOfChange : WORD;	
	{attribute 'OPC.UA.DA' := '1'}
	PV7 AT %M* : UINT;  //Antal minuter insamlade för medelvärdesberäkning (max 4320)~wp:[unit]minuter[format]0
	{attribute 'OPC.UA.DA' := '1'}
	OPM AT %M* : REAL;//Värde handställning~wp:[unit]°C[format]0.0
	{attribute 'OPC.UA.DA' := '1'}
	SP1 AT %M* : UINT := 12; //Antal timmar för medelvärdesberäkning (2-72)~wp:[unit]timmar[format]0
	
	rArrayMean72Hours : ARRAY [0..4319] OF REAL;
	tAlarmDelayDifferenceCheck : TIME := T#48H;
END_VAR

	// Kollar så värdet uppdateras från överliggande system
	fbDifferenceCheckTemp(rPv:=PV );
	fbAlarmTemp(bInput:= NOT fbDifferenceCheckTemp.bDifference , tAlarmDelay:=tAlarmDelayDifferenceCheck , bAutoReset:=TRUE , bAlarmOutput=>FAULT);
	
	IF bResetMeanTemp THEN
		bResetMeanTemp := FALSE;
		PV7 := 2;
	END_IF

	IF SP1 > 72 THEN // Medelvärdestid maxbegränsas till 72 timmar.
		SP1 := 72;
	ELSIF SP1 < 2 THEN // Medelvärdestid minbegränsas till 2 timmar.
		SP1 := 2;
	END_IF
	
	IF SP1 <= 72 AND SP1 > 1 THEN
		 iAntalMinuterMedel := SP1 * 60;
	END_IF;

	mMean(); // Metod för att räkna ut medelvärde
	//4320 minuter = 72 timmar.
	IF iAntalMinuterForUtrakning > 2 THEN
		PV1 := LREAL_TO_REAL(lrMeanInternal) / iAntalMinuterForUtrakning; 
	END_IF;
	
	oaksGVL.rOutdoorTemp := PV; //utetemp som behåller sitt senaste giltiga värde vid givarfel 
	
	IF NOT FAULT THEN 
		oaksGVL.rOutdoorTempErrorValue0 := PV; // global utetemp som ställs till 0 vid givarfel.
		oaksGVL.rOutdoorTempErrorValue150 := PV;// global utetemp som ställs till 150 vid givarfel.
	ELSE
		oaksGVL.rOutdoorTempErrorValue0 := 0; // global utetemp som ställs till 0 vid givarfel.
		oaksGVL.rOutdoorTempErrorValue150 := 150;// global utetemp som ställs till 150 vid givarfel.
	END_IF
	oaksGVL.rOutdoorTempMean := PV1; // global medel utetemp
	
	oaksGVL.bOutdoorTempSensorError := FAULT; // globalt utegivarfel

METHOD PRIVATE mMean : BOOL // metod för att sköta uträkning av medelvärde
VAR_INPUT
END_VAR
	FB_BA_GetTime01(bEn :=TRUE);	
	stTime := FB_BA_GetTime01.stSysTi;

	IF stTime.wMinute <> wLastMinuteOfChange THEN
		fbMinuteTrig(CLK := TRUE);
	ELSE
		fbMinuteTrig(CLK := FALSE);
	END_IF
	//4320 minuter - 1 = 72 timmar.
	IF fbMinuteTrig.Q THEN
		FOR iCounter:= iAntalMinuterMedel - 1 TO 1 BY -1 DO
			rArrayMean72Hours[iCounter]:=rArrayMean72Hours[iCounter-1];
		END_FOR;
		rArrayMean72Hours[0] := PV;
		wLastMinuteOfChange := stTime.wMinute;
		IF PV7 < 4320 THEN // Räknas upp för att hålla koll på antal insamlade minuter
			PV7 := PV7 +1;
		END_IF
	END_IF 
	
	lrMeanInternal := 0;
	//4320 minuter - 1 = 72 timmar.
	iAntalMinuterForUtrakning := MIN(iAntalMinuterMedel,PV7); // Max begränsar antal minuter som används för beräkning beroende på hur många minuter som finns insamlade
	FOR iCounter:= iAntalMinuterForUtrakning TO 1 BY -1 DO
		lrMeanInternalTemp := lrMeanInternal;
		lrMeanInternal:=rArrayMean72Hours[iCounter-1] + lrMeanInternalTemp;
	END_FOR;
END_METHOD

END_FUNCTION_BLOCK

// oaksLibrary/Larm/Larm med inbyggd larmtagg/fbFreezeAlarm
//Frysvaktsblock med integrerad handställbar pt1000-givare. Handställning förreglas om insignal underskrider 12 grader eller vid givarfel.
//Minbegränsning returtemperatur vid drift stopp aggregat går ej att ställa under 10°C.
FUNCTION_BLOCK fbFreezeAlarm EXTENDS fbPT1000
VAR_INPUT
	bOperationIndication : BOOL; // Driftindikering för tilluftsfläkt kopplas hit. Används för att avgöra vilket minbegränsningsbörvärde som skall användas.
END_VAR
VAR_OUTPUT
	{attribute 'OPC.UA.DA' := '1'}
	LAL AT %M* : BOOL; //Frysvakt~wp:[alarmoptions]p:1,rst:OAKSGVL_RST=1
	rMinOutput : REAL; // Utsignal minbegränsning returvattenregulator 
END_VAR
VAR
	fbReg01 : Tc3_BA_Common.FB_BA_PIDCtrl;
	rSetpoint : REAL;
	fbFreezeInterlock : fbAlarm;
	//itemp :INT;
	{attribute 'OPC.UA.DA' := '1'}
	PV8 AT %M* : REAL; //Aktuell reglersignal minbegränsningsregulator~wp:[unit]%[format]0[trendoptions]i:300
END_VAR
VAR_INPUT PERSISTENT
	{attribute 'OPC.UA.DA' := '1'}
	ALL AT %M* : REAL := 7; //Larmgräns frysvakt~wp:[unit]°C[format]0.0
	{attribute 'OPC.UA.DA' := '1'}
	SP1 AT %M* : REAL := 12; //Minbegränsning returtemperatur vid drift av aggregat~wp:[unit]°C[format]0.0
	{attribute 'OPC.UA.DA' := '1'}
	SP2 AT %M* : REAL := 15; //Minbegränsning returtemperatur vid drift stopp av aggregat~wp:[unit]°C[format]0.0
END_VAR

	SUPER^();

	//Handställning förreglas om insignal underskrider 12 grader eller vid givarfel
	IF FB_BA_AI01.rVal < 12 OR FAULT THEN
		M := FALSE;
	END_IF
	
	// Minbegränsning av frysvaktsinställning 5 grader
	IF ALL < 5.0 THEN 
		ALL := 5.0;
	END_IF

	
	// Frysvaktslarm om temperatur underskrider inställt värde. 
	fbFreezeInterlock(
	bInput:= PV < ALL OR FAULT, 
	tAlarmDelay:= T#3S , 
	bAutoReset:=FALSE , 
	bAlarmOutput=> LAL);
	
	
	// Minbegränsning av inställningsvärde för returtemperatur vid stopp av aggregat
	IF SP2 < 10.0 THEN 
		SP2 := 10.0;
	END_IF
	// Val av börvärde till minbegränsningsregulator
	IF bOperationIndication THEN
		rSetpoint := SP1;
	ELSE
		rSetpoint := SP2;
	END_IF
	
	fbReg01(
	bEn:=TRUE , 
	rW:=rSetpoint , 
	rX:=PV , 
	udiOpMode:= , 
	bActn:= , 
	rKp:= 20, 
	udiTn_ms:= , 
	udiTv_ms:= , 
	udiTd_ms:= , 
	rYMax:=100 , 
	rYMin:= 0, 
	rNZ:= , 
	udiCycCl:= , 
	bSync:= , 
	rSync:= , 
	rY=> , 
	rE=> , 
	bARW=> );
	
	IF NOT FAULT THEN
		rMinOutput := fbReg01.rY;
	ELSE
		rMinOutput := 100;
	END_IF
	// För visning och trendning i webport
	PV8 := rMinOutput;

END_FUNCTION_BLOCK

// oaksLibrary/Larm/Larm med inbyggd larmtagg/fbFreezeAlarmVoltage
//Frysvaktsblock med integrerad handställbar aktiv givare. Handställning förreglas om insignal underskrider 12 grader eller vid givarfel.
//Minbegränsning returtemperatur vid drift stopp aggregat går ej att ställa under 10°C.
FUNCTION_BLOCK fbFreezeAlarmVoltage EXTENDS fbVoltageTemp
VAR_INPUT
	bOperationIndication : BOOL; // Driftindikering för tilluftsfläkt kopplas hit. Används för att avgöra vilket minbegränsningsbörvärde som skall användas.

END_VAR
VAR_OUTPUT
	{attribute 'OPC.UA.DA' := '1'}
	LAL AT %M* : BOOL; //Frysvakt~wp:[alarmoptions]p:1,rst:OAKSGVL_RST=1
	rMinOutput : REAL; // Utsignal minbegränsning returvattenregulator 
END_VAR
VAR
	fbReg01 : Tc3_BA_Common.FB_BA_PIDCtrl;
	rSetpoint : REAL;
	fbFreezeInterlock : fbAlarm;
	//itemp :INT;
	{attribute 'OPC.UA.DA' := '1'}
	PV7 AT %M* : REAL; //Aktuell reglersignal minbegränsningsregulator~wp:[unit]%[format]0[trendoptions]i:300
END_VAR
VAR_INPUT PERSISTENT
	{attribute 'OPC.UA.DA' := '1'}
	ALL AT %M* : REAL := 7; //Larmgräns frysvakt~wp:[unit]°C[format]0.0
	{attribute 'OPC.UA.DA' := '1'}
	SP1 AT %M* : REAL := 12; //Minbegränsning returtemperatur vid drift av aggregat~wp:[unit]°C[format]0.0
	{attribute 'OPC.UA.DA' := '1'}
	SP2 AT %M* : REAL := 15; //Minbegränsning returtemperatur vid drift stopp av aggregat~wp:[unit]°C[format]0.0
END_VAR

	SUPER^();

	//Handställning förreglas om insignal underskrider 12 grader eller vid givarfel
	IF FB_BA_AI01.rVal < 12 OR FAULT THEN
		M := FALSE;
	END_IF
	
	// Minbegränsning av frysvaktsinställning 5 grader
	IF ALL < 5.0 THEN 
		ALL := 5.0;
	END_IF

	
	// Frysvaktslarm om temperatur underskrider inställt värde. 
	fbFreezeInterlock(
	bInput:= PV < ALL OR FAULT, 
	tAlarmDelay:= T#3S , 
	bAutoReset:=FALSE , 
	bAlarmOutput=> LAL);
	
	
	// Minbegränsning av inställningsvärde för returtemperatur vid stopp av aggregat
	IF SP2 < 10.0 THEN 
		SP2 := 10.0;
	END_IF
	// Val av börvärde till minbegränsningsregulator
	IF bOperationIndication THEN
		rSetpoint := SP1;
	ELSE
		rSetpoint := SP2;
	END_IF
	
	fbReg01(
	bEn:=TRUE , 
	rW:=rSetpoint , 
	rX:=PV , 
	udiOpMode:= , 
	bActn:= , 
	rKp:= 20, 
	udiTn_ms:= , 
	udiTv_ms:= , 
	udiTd_ms:= , 
	rYMax:=100 , 
	rYMin:= 0, 
	rNZ:= , 
	udiCycCl:= , 
	bSync:= , 
	rSync:= , 
	rY=> , 
	rE=> , 
	bARW=> );
	
	IF NOT LAL THEN
		rMinOutput := fbReg01.rY;
	ELSE
		rMinOutput := 100;
	END_IF

	// För visning och trendning i webport
	PV7 := rMinOutput;

END_FUNCTION_BLOCK

// oaksLibrary/Larm/Larm med inbyggd larmtagg/fbFusealarm
FUNCTION_BLOCK fbFusealarm
VAR_INPUT
	{attribute 'OPC.UA.DA' := '1'}
	V3 AT %I* : BOOL; //Larmingång~wp:[trendoptions]i:14400, t:1
	bInvert : BOOL;
	bAutoReset : BOOL := TRUE; // Auto-reset av larm
END_VAR
VAR_OUTPUT
	{attribute 'OPC.UA.DA' := '1'}
	AL AT %M*  : BOOL; //Utlöst automatsäkring~wp:
END_VAR
VAR
	bInternalIndication : BOOL;
	fbAlarm1 : fbAlarm;
END_VAR

	IF NOT bInvert THEN
		bInternalIndication :=  V3;
	ELSE
		bInternalIndication := NOT V3;
	END_IF
		
	
	fbAlarm1(
	bInput:= bInternalIndication, 
	tAlarmDelay:= T#500MS, 
	bAutoReset:= bAutoReset, 
	bAlarmOutput=>AL );

END_FUNCTION_BLOCK

// oaksLibrary/Larm/Larm med inbyggd larmtagg/fbJfb
FUNCTION_BLOCK fbJfb
VAR_INPUT
	{attribute 'OPC.UA.DA' := '1'}
	V3 AT %I* : BOOL; //Larmingång~wp:[trendoptions]i:14400, t:1
	bInvert : BOOL;
	bAutoReset : BOOL := TRUE; // Auto-reset av larm
END_VAR
VAR_OUTPUT
	{attribute 'OPC.UA.DA' := '1'}
	AL AT %M*  : BOOL; //Utlöst jordfelsbrytare~wp:
END_VAR
VAR
	bInternalIndication : BOOL;
	fbAlarm1 : fbAlarm;
END_VAR

	IF NOT bInvert THEN
		bInternalIndication :=  V3;
	ELSE
		bInternalIndication := NOT V3;
	END_IF
		
	
	fbAlarm1(
	bInput:= bInternalIndication, 
	tAlarmDelay:= T#500MS, 
	bAutoReset:= bAutoReset, 
	bAlarmOutput=>AL );

END_FUNCTION_BLOCK

// oaksLibrary/Larm/Larm med inbyggd larmtagg/fbLeakDetector
//OAKS AB
//2021-02-08
//Funktionsblock för beräkning av läckage i tex. kallvattensystem
//Funktionen är aktiv mellan inställt intervall för start-/stopptimme (stopptimme avser den timme då funktion stoppar om tex timme 5 ställs stoppar funktion då timme slår om till 5).
//Om inte 0-flöde uppmäts då funktion är aktiv under enligt inställda värden utgår larm.

FUNCTION_BLOCK fbLeakDetector
VAR_INPUT
	iHour : INT; //Aktuell timme
	rVolume : REAL; //Mätarställning från mätare
END_VAR

VAR_INPUT PERSISTENT
	{attribute 'OPC.UA.DA' := '1'}
	SP1 AT %M* : INT := 3; //Starttimme beräkning~wp:[format]0
	{attribute 'OPC.UA.DA' := '1'}
	SP2 AT %M* : INT := 5; //Stopptimme beräkning~wp:[format]0
	{attribute 'OPC.UA.DA' := '1'}
	AHL AT %M* : INT := 3; //Larmgräns antal dagar med fel~wp:[format]0
	{attribute 'OPC.UA.DA' := '1'}
	AD AT %M* : REAL := 5; //Samplingstid nollförbrukning~wp:[format]0[unit]min
END_VAR

VAR_OUTPUT
	{attribute 'OPC.UA.DA' := '1'}
	PV1 AT %M* : INT; //Antal dagar med fel~wp:[format]0
	{attribute 'OPC.UA.DA' := '1'}
	PV8 AT %M* : REAL; //Aktuell differens~wp:[format]0
	{attribute 'OPC.UA.DA' := '1'}
	V AT %M* : BOOL; //Beräkning aktiv~wp:[trendoptions]i:14400, t:1
	{attribute 'OPC.UA.DA' := '1'}
	AL AT %M* : BOOL; //Läckagelarm~wp:[alarmoptions]P:2
END_VAR
VAR
	rNewValue : REAL := 0;
	rStoredValue : REAL := 0;
	bZeroValueOk : BOOL;
	TON_zero : TON;
	F_TRIG_CalcFinished: F_TRIG;
	fbAlarm_Fault : fbAlarm;
	TON_Sampler: TON;
	bReset : BOOL := FALSE;
END_VAR

//Samplingstid
TON_Sampler(IN:= NOT bReset, PT:= T#5S, Q=> , ET=> );
	
	bReset := FALSE;
	
	//Om värden skiljer sig åt
	IF TON_Sampler.Q THEN
		PV8 := rVolume - rStoredValue;	
		rStoredValue := rVolume;
		bReset := TRUE;
	END_IF;

//Starta beräkning 
IF iHour >= SP1 AND iHour < SP2 THEN
	V := TRUE;
ELSE
	//När beräkning ej är aktiv
	V := FALSE; 
END_IF
	
//Beräkning ingen förbrukning under 5 minuter
TON_zero(IN:= (PV8 = 0) AND V,PT:=REAL_TO_TIME(AD*60000) , Q=> , ET=> );

IF TON_zero.Q THEN
	bZeroValueOk := TRUE;
END_IF

//Räkna upp antal dagar det varit fel
F_TRIG_CalcFinished(CLK:= V, Q=> );

IF F_TRIG_CalcFinished.Q AND NOT bZeroValueOk THEN
	PV1 := PV1 + 1;
	//Återställ att värdet är ok inför nästa dag
	bZeroValueOk := FALSE;
ELSIF F_TRIG_CalcFinished.Q AND bZeroValueOk THEN
	PV1 := 0;
	//Återställ att värdet är ok inför nästa dag
	bZeroValueOk := FALSE;
END_IF

//Alarm då antal dagar uppnåtts
fbAlarm_Fault(bInput:= PV1 >= AHL, tAlarmDelay:= T#5S, bAutoReset:= TRUE, bAlarmOutput=> );
AL := fbAlarm_Fault.bAlarmOutput;

END_FUNCTION_BLOCK

// oaksLibrary/Larm/Larm med inbyggd larmtagg/fbManometerLow
FUNCTION_BLOCK fbManometerLow
VAR_INPUT
	{attribute 'OPC.UA.DA' := '1'}
	V3 AT %I* : BOOL; //Larmingång låglarm~wp:[trendoptions]i:14400, t:1
	bInvertLow : BOOL;
	bAutoReset : BOOL := TRUE; // Auto-reset av larm
END_VAR
VAR_OUTPUT
	{attribute 'OPC.UA.DA' := '1'}
	AL AT %M*  : BOOL; //Lågt tryck~wp:
END_VAR
VAR
	bInternalIndicationLow : BOOL;
	fbAlarm1 : fbAlarm;
END_VAR
VAR_INPUT PERSISTENT
	{attribute 'OPC.UA.DA' := '1'}
	AD AT %M*  : REAL := 30; //Larmfördröjning~wp:[unit]sekunder
END_VAR

	IF NOT bInvertLow THEN
		bInternalIndicationLow :=  V3;
	ELSE
		bInternalIndicationLow := NOT V3;
	END_IF
		
	fbAlarm1(
	bInput:= bInternalIndicationLow, 
	tAlarmDelay:= fRealToSecond(rSecond:=AD ), 
	bAutoReset:= bAutoReset, 
	bAlarmOutput=>AL );

END_FUNCTION_BLOCK

// oaksLibrary/Larm/Larm med inbyggd larmtagg/fbManometerLowHigh
FUNCTION_BLOCK fbManometerLowHigh EXTENDS fbManometerLow
VAR_INPUT
	{attribute 'OPC.UA.DA' := '1'}
	V4 AT %I* : BOOL; //Larmingång höglarm~wp:[trendoptions]i:14400, t:1
	bInvertHigh : BOOL;
END_VAR
VAR_OUTPUT
	{attribute 'OPC.UA.DA' := '1'}
	AL1 AT %M*  : BOOL; //Högt tryck~wp:
END_VAR
VAR
	bInternalIndicationHigh : BOOL;
	fbAlarm2 : fbAlarm;
END_VAR

	SUPER^();
	
	IF NOT bInvertHigh THEN
		bInternalIndicationHigh :=  V4;
	ELSE
		bInternalIndicationHigh := NOT V4;
	END_IF
		
	fbAlarm2(bInput:=bInternalIndicationHigh , 
	tAlarmDelay:=fRealToSecond(rSecond:=AD ) , 
	bAutoReset:= bAutoReset,
	bAlarmOutput=>AL1 );

END_FUNCTION_BLOCK

// oaksLibrary/Larm/Larm med inbyggd larmtagg/fbOvervoltageProtection
FUNCTION_BLOCK fbOvervoltageProtection
VAR_INPUT
	{attribute 'OPC.UA.DA' := '1'}
	V3 AT %I* : BOOL; //Larmingång~wp:[trendoptions]i:14400, t:1
	bInvert : BOOL;
	bAutoReset : BOOL := TRUE; // Auto-reset av larm
END_VAR
VAR_OUTPUT
	{attribute 'OPC.UA.DA' := '1'}
	AL AT %M*  : BOOL; //Utlöst överspänningsskydd~wp:
END_VAR
VAR
	bInternalIndication : BOOL;
	fbAlarm1 : fbAlarm;
END_VAR

	IF NOT bInvert THEN
		bInternalIndication :=  V3;
	ELSE
		bInternalIndication := NOT V3;
	END_IF
		
	
	fbAlarm1(
	bInput:= bInternalIndication, 
	tAlarmDelay:= T#500MS, 
	bAutoReset:= bAutoReset, 
	bAlarmOutput=>AL );

END_FUNCTION_BLOCK

// oaksLibrary/Larm/Larm med inbyggd larmtagg/fbRotationGuard
// Block för rotationsvaktslarm VVX.
FUNCTION_BLOCK fbRotationGuard
VAR_INPUT
	rSetpoint : REAL;//Ingång vvx-utsignal
	{attribute 'OPC.UA.DA' := '1'}
	V3 AT %I* : BOOL; //Ingång rotationsvakt~wp:
	bAutoReset : BOOL := TRUE; // Auto-reset av larm
END_VAR
VAR_OUTPUT
	{attribute 'OPC.UA.DA' := '1'}
	AL AT %M*  : BOOL; //Rotationsvakt värmeväxlare~wp:
END_VAR
VAR
	fbAlarm1 : fbAlarm;
	
	fbTonOn : TON;
	fbTonOff : TON;
END_VAR
VAR PERSISTENT
	{attribute 'OPC.UA.DA' := '1'}
	AD AT %M* : REAL := 5; //Larmfördröjning rotationsvakt~wp:[format]0[unit]min
END_VAR

	fbTonOn(IN:= V3 AND rSetpoint = 100, PT:=fRealToMinute(AD)  , Q=> , ET=> );
	fbTonOff(IN:= NOT V3 AND rSetpoint = 100, PT:=fRealToMinute(AD)  , Q=> , ET=> );

	fbAlarm1(
	bInput:= fbTonOn.Q OR fbTonOff.Q, 
	tAlarmDelay:= T#3S, 
	bAutoReset:= bAutoReset, 
	bAlarmOutput=>AL );

END_FUNCTION_BLOCK

// oaksLibrary/Larm/fbDamperAlarmOneInput
// funktionsblock för spjäll-lägeslarm för spjäll med en indikering. Larmar om bDamperOutput är till och bDamperInput inte är till.
FUNCTION_BLOCK fbDamperAlarmOneInput
VAR_INPUT
	bDamperOutput : BOOL;// hit knyts spjällets utsignal
	bDamperInput : BOOL; // hit knyts spjällets indikering
	tAlarmDelay : TIME := T#180S; // Larmfördröjning
	bAutoReset : BOOL; // Ange om larmet ska vara autoresetande.
END_VAR
VAR_OUTPUT
	bDamperAlarm : BOOL; // Larm utgång spjäll i fel läge
END_VAR
VAR
	fbAlarmDelay : TON;
	fbDamperAlarm : fbAlarm; 
END_VAR

fbAlarmDelay(IN:=bDamperOutput AND NOT bDamperInput  , PT:=tAlarmDelay , Q=> , ET=> );

fbDamperAlarm(bInput:= fbAlarmDelay.Q , tAlarmDelay:=T#0S , bAutoReset:=bAutoReset , bAlarmOutput=>bDamperAlarm );

END_FUNCTION_BLOCK

// oaksLibrary/Larm/fbDevAlarm
// Avvikelselarm 
FUNCTION_BLOCK fbDevAlarm EXTENDS fbAlarm
VAR_INPUT
	bEnable : BOOL; // FALSE = larm blockerat
	rProcessValue : REAL; // Ärvärde
	rSetPoint : REAL; // Larmgräns
	rDevLimit : REAL;
	bBlockHighAlarm : BOOL; // Blockera högtemplarm
	bBlockLowAlarm : BOOL; // Blockera lågtemplarm
END_VAR
VAR_OUTPUT
END_VAR
VAR
		iTemp1: INT;
END_VAR

	SUPER^();

	IF rProcessValue > (rSetPoint + rDevLimit) AND bEnable AND NOT bBlockHighAlarm THEN
		bInput := TRUE;
	ELSIF rProcessValue < (rSetPoint - rDevLimit) AND bEnable AND NOT bBlockLowAlarm THEN
		bInput := TRUE;
	ELSE	
		bInput := FALSE;
	END_IF;

END_FUNCTION_BLOCK

// oaksLibrary/Larm/fbDigitalAlarmIO
// Larmblock för digitala larm. Inbyggda taggar för ingång och fördröjning. 
FUNCTION_BLOCK fbDigitalAlarmIO
VAR_INPUT
	{attribute 'OPC.UA.DA' := '1'}
	V3 AT %I* : BOOL; //Larmingång~wp:[trendoptions]i:14400, t:1
	bInvert : BOOL;
	bAutoReset : BOOL := TRUE; // Auto-reset av larm
	bEnable : BOOL := TRUE; 
END_VAR
VAR_OUTPUT
	bOutput : BOOL;
END_VAR
VAR
	bInternalIndication : BOOL;
	fbAlarm1 : fbAlarm;
END_VAR
VAR_INPUT PERSISTENT
	{attribute 'OPC.UA.DA' := '1'}
	AD AT %M* : REAL := 3; //Larmfördröjning~wp:[unit]sekunder[format]0
END_VAR

	IF NOT bInvert THEN
		bInternalIndication :=  V3;
	ELSE
		bInternalIndication := NOT V3;
	END_IF
		
	
	fbAlarm1(
	bInput:= bInternalIndication AND bEnable, 
	tAlarmDelay:= REAL_TO_TIME(AD*1000), 
	bAutoReset:= bAutoReset, 
	bAlarmOutput=>bOutput );

END_FUNCTION_BLOCK

// oaksLibrary/Larm/fbFloorheatHighTemp
//Oaks AB
//2021-09-06
//Funktionsblock för blockering av golvvärme vid hög framledningstemperatur. Då temperatur överstiger inställt värde under 5min blockeras pump i 15 min, funktionen återstartar efter 15min. 
FUNCTION_BLOCK fbFloorheatHighTemp
VAR_INPUT
	rProcessValue : REAL := 3; //Golvvärmetemperatur
	rHighLimit : REAL := 45; //Stopp temperatur
	rLowLimit : REAL := 40; //Start temperatur
END_VAR
VAR_OUTPUT
	bPumpStart : BOOL; //Pumpblockering (True då förregling ej är aktiv)
	PV1 AT %M* : STRING := ' '; //Driftinformation~wp:
	PV8 AT %M* : STRING := ' '; //Konfigurering~wp:
END_VAR
VAR
	fbHystReal_Start : fbHystReal;
	fbTON_StopDelay: TON;
	fbTOF_StopDelay : TOF;
	sTemp : STRING := '';
	sTemp1 : STRING := '';
	sTemp2 : STRING := '';
	rTemp : REAL := 0;
	tSetStopDelTime: TIME;
END_VAR

//Blockering hysteres
fbHystReal_Start(rPv:= rProcessValue, rHigh:= rHighLimit, rLow:= rLowLimit, bOutput=> );

//Fördröjning innan stopp
IF fbHystReal_Start.bOutput THEN
	tSetStopDelTime := T#15M;
ELSE
 	tSetStopDelTime := T#0S;
END_IF

fbTON_StopDelay(IN:= fbHystReal_Start.bOutput AND NOT fbTOF_StopDelay.Q, PT:= T#5M, Q=> , ET=> );

IF fbHystReal_Start.bOutput THEN
	fbTOF_StopDelay(IN:= fbTON_StopDelay.Q, PT:= tSetStopDelTime, Q=> , ET=> );
ELSE 
	fbTOF_StopDelay(IN:=FALSE, PT:= tSetStopDelTime, Q=> , ET=> );
END_IF

//Blockering pump
bPumpStart := NOT fbTOF_StopDelay.Q;

//Statustexter
rTemp := (TIME_TO_REAL(fbTOF_StopDelay.PT) - TIME_TO_REAL(fbTOF_StopDelay.ET)) / 1000;
sTemp := LREAL_TO_FMTSTR(rTemp, 0, TRUE );
sTemp := CONCAT('Pump blockerad, återstående tid ', sTemp);
sTemp := CONCAT(sTemp, ' sekunder');

IF bPumpStart THEN
	PV1 := ' ';
ELSE
	PV1 := sTemp;
END_IF

sTemp1 := CONCAT('Hög gräns: ',REAL_TO_STRING(rHighLimit));
sTemp1 := CONCAT(sTemp1, ' C°');
sTemp2 := CONCAT('<br>Låg gräns: ',REAL_TO_STRING(rLowLimit));
sTemp2 := CONCAT(sTemp2, ' C°');	
PV8 := CONCAT(sTemp1,sTemp2);

END_FUNCTION_BLOCK

// oaksLibrary/fbHystReal
//Funktionsblock för hysteres. bOutput går till då rPv är större än rHigh och från då rPv är lägre än rLow.
FUNCTION_BLOCK fbHystReal
VAR_INPUT
rPv : REAL; //Ärvärde
rHigh : REAL; //Hög gräns
rLow : REAL; //Låg gräns
END_VAR
VAR_OUTPUT
bOutput : BOOL :=FALSE; //Utgång
END_VAR
VAR
END_VAR

IF rPV >= rHigh THEN
	bOutput := TRUE;
ELSIF  rPv <= rLow THEN
	bOutput := FALSE;
END_IF

END_FUNCTION_BLOCK

// oaksLibrary/Larm/fbFreezeAlarmNoSensor
//Frysvaktsblock utan inbyggd givare (för användning med t ex modbus-givare)
//Minbegränsning returtemperatur vid drift stopp aggregat går ej att ställa under 10°C.
FUNCTION_BLOCK fbFreezeAlarmNoSensor
VAR_INPUT
	bOperationIndication : BOOL; // Driftindikering för tilluftsfläkt kopplas hit. Används för att avgöra vilket minbegränsningsbörvärde som skall användas.
	rPV	: REAL;	//Mätvärde givare
	bFAULT : BOOL; //Givarfel
	
	rALL AT %M* : REAL := 7; //Larmgräns frysvakt
	rSP1 AT %M* : REAL := 12; //Minbegränsning returtemperatur vid drift av aggregat
	rSP2 AT %M* : REAL := 15; //Minbegränsning returtemperatur vid drift stopp av aggregat
END_VAR
VAR_OUTPUT
	bLAL : BOOL; //Frysvakt
	rMinOutput : REAL; //Utsignal minbegränsning returvattenregulator 
END_VAR
VAR
	fbReg01 : Tc3_BA_Common.FB_BA_PIDCtrl;
	rSetpoint : REAL;
	fbFreezeInterlock : fbAlarm;
END_VAR
VAR_INPUT PERSISTENT
END_VAR

// Minbegränsning av frysvaktsinställning 5 grader
	IF rALL < 5.0 THEN 
		rALL := 5.0;
	END_IF
	
// Frysvaktslarm om temperatur underskrider inställt värde. 
	fbFreezeInterlock(
	bInput:= rPV < rALL OR bFAULT, 
	tAlarmDelay:= T#3S , 
	bAutoReset:=FALSE , 
	bAlarmOutput=> bLAL);
	
// Minbegränsning av inställningsvärde för returtemperatur vid stopp av aggregat
	IF rSP2 < 10.0 THEN 
		rSP2 := 10.0;
	END_IF
	// Val av börvärde till minbegränsningsregulator
	IF bOperationIndication THEN
		rSetpoint := rSP1;
	ELSE
		rSetpoint := rSP2;
	END_IF
	
	fbReg01(
	bEn:=TRUE , 
	rW:=rSetpoint , 
	rX:=rPV , 
	udiOpMode:= , 
	bActn:= , 
	rKp:= 20, 
	udiTn_ms:= , 
	udiTv_ms:= , 
	udiTd_ms:= , 
	rYMax:=100 , 
	rYMin:= 0, 
	rNZ:= , 
	udiCycCl:= , 
	bSync:= , 
	rSync:= , 
	rY=> , 
	rE=> , 
	bARW=> );
	
	IF NOT bLAL THEN
		rMinOutput := fbReg01.rY;
	ELSE
		rMinOutput := 100;
	END_IF

END_FUNCTION_BLOCK

// oaksLibrary/Mätare/fbEnergyCounterCondition
//Samplar energiräknare från en annan källa (t ex energimätare via mbus etc), för att beräkna förbrukad energi när ingångsvillkor är till.
//Kan t ex användas för att beräkna energiförbrukning från en mätare endast när en tidkanal är till
//Testad 231120
//Robert H, 231120 
FUNCTION_BLOCK fbEnergyCounterCondition
VAR_INPUT
	rEnergyIn	: REAL;				//Energivärde från extern källa
	bCondition	: BOOL;				//Villkor för att beräkna förbrukning i detta block
	bReset		: BOOL := FALSE;	//Återställ räknare (OBS måste inkomma 2ggr inom 30 sekunder för att utföras)
END_VAR
VAR_OUTPUT PERSISTENT
	rEnergyCondition : REAL;		//Energiförbrukning när bCondition varit till
END_VAR
VAR
	fbConditionEdge	: fbEdge;
	rEnergySampleStart	: REAL;
	rEnergySampleStop	: REAL;
	byResetCnt			: BYTE;
	bResetTOF			: TOF;
END_VAR

//Övervaka villkor för beräkning
fbConditionEdge(anyInput := bCondition);

//Om villkor går till, sampla aktuellt energivärde
IF fbConditionEdge.bEdgeF AND bCondition THEN
	rEnergySampleStart := rEnergyIn;
//Om villkor går från, sampla aktuellt energivärde igen och summera diff på räknarvariabel
ELSIF fbConditionEdge.bEdgeF AND NOT bCondition THEN
	rEnergySampleStop := rEnergyIn;
	rEnergyCondition := rEnergyCondition + (rEnergySampleStop - rEnergySampleStart);
END_IF;

//Återställningsfunktion; starta timer när bReset inkommit. Om bReset inkommer en gång till inom timertiden, utför återställning	
bResetTOF(IN := bReset, PT := T#30S);

IF bResetTOF.Q AND bReset THEN
	byResetCnt := byResetCnt + 1;
	bReset := FALSE;
	
	IF byResetCnt >= 2 THEN
		rEnergyCondition := 0;
		byResetCnt := 0;
	END_IF
END_IF

IF NOT bResetTOF.Q THEN
	byResetCnt := 0;
END_IF

END_FUNCTION_BLOCK

// oaksLibrary/Mätare/fbPulseMeterE_P
//Pulsräknare för beräkning av energi samt momentan effekt med tidsfaktor och remanens
//Blocket är enhetsagnostiskt. För att få önskad enhet kan du antingen ställa in pulsfaktor så att det motsvarar den enhet du önskar:
//	- t ex om mätaren pulsar Wh och du vill ha kW ställer du pulsfaktor på 0.001
//Eller så kan du ställa pulsfaktorn på 1, blocket kommer då räkna Wh, sen kan du dela utvariabeln rEnergy med 1000 för att få önskad enhet.
//Vill du ha olika storhet på räknaren (t ex energi) och momentana värdet (t ex effekt) får du använda båda metoderna:
// - t ex för att få energi i MWh och effekt i kWh och mätaren pulsar kWh, så ställer du pulsfaktorn till 0.001. Sen gångrar du rPower med 1000.
//Samplingstid på 60s funkar i de flesta fall. Remanens används för att undvika att det momentana värdet faller till 0 direkt om det går längre tid än samplingstiden mellan pulser.
//Manuell omställning av mätaren kan göras på SP1. Ställ värdet till minst 1 (0 kommer ej att uppdatera räknaren)
//OAKS, 23-10-31

FUNCTION_BLOCK fbPulseMeterE_P
VAR_INPUT
	bPulse AT %I* : BOOL; //Pulsingång~wp:
	{attribute 'OPC.UA.DA' := '1'}
	SP1 AT %M* : LREAL := 1; //Nytt värde mätarställning (obs lägst 1)~wp:[format]0.000
END_VAR

VAR_OUTPUT
	lrEnergy	: LREAL; //Energi
	rPower  : REAL; //Beräknad effekt
	{attribute 'OPC.UA.DA' := '1'}
	PV5 AT %M* : INT; //Klockslag vid senaste puls (12:01 visas som 1201)~wp:
	{attribute 'OPC.UA.DA' := '1'}
	FAULT  AT %M* : BOOL; //Samplingstid/pulsfaktor får ej vara 0~wp:
END_VAR
VAR
	stTime		: tc2_ba.TIMESTRUCT;
	nActualDayCase	: INT;
	nActualHour 	: INT;
	nActualMinute 	: INT;
	
	FB_BA_GetTime01 : tc2_ba.FB_BA_GetTime; 		

	fbCounterTrig : r_trig;
	
	ulInternalStorageValueOld : ULINT;
	
	fbPowerCalcTimer : TON;
	ulDeltaEnergy : ULINT;
	fbRemTimer : TON;	
	fbEdgeEn : fbEdge;
END_VAR
VAR PERSISTENT 
	ulInternalStorageValue : ULINT; // Internt värde
END_VAR
VAR_INPUT PERSISTENT
	{attribute 'OPC.UA.DA' := '1'}
	SP2 AT %M* : REAL := 1; //Pulsfaktor (t ex 0.001 för kWh om mätarens pulsenhet är Wh)~wp:
	{attribute 'OPC.UA.DA' := '1'}
	SP3 AT %M* : UDINT := 60; //Samplingstid för effektberäkning~wp:[unit]s[format]0
	{attribute 'OPC.UA.DA' := '1'}
	SP4 AT %M* : UDINT := 0; //Remanens för effektberäkning~wp:[unit]s[format]0
END_VAR

IF SP3 = 0 THEN
	SP3 := 1;
END_IF

IF SP2 = 0 THEN
	SP3 := 1;
END_IF

FAULT := (SP2 = 0) OR (SP3 = 0);

//Beräkning energi
FB_BA_GetTime01(bEn :=TRUE);	
stTime := FB_BA_GetTime01.stSysTi;

nActualDayCase :=WORD_TO_INT (stTime.wDayOfWeek);
nActualHour :=WORD_TO_INT (stTime.wHour)*100;
nActualMinute :=WORD_TO_INT (stTime.wMinute);

fbCounterTrig(CLK:=bPulse , Q=> );

IF fbCounterTrig.Q THEN 
	ulInternalStorageValue := ulInternalStorageValue + 1;
	PV5 := nActualHour+nActualMinute;
END_IF

lrEnergy := ULINT_TO_LREAL(ulInternalStorageValue) * SP2;

fbEdgeEn(anyInput := SP1);

IF fbEdgeEn.bEdgeF AND SP1 <> 0 THEN
	ulInternalStorageValue := LREAL_TO_ULINT(SP1 / SP2);
	SP1 := 0;
 	ulInternalStorageValueOld := ulInternalStorageValue;
END_IF

//Beräkning effekt
fbPowerCalcTimer(PT := UDINT_TO_TIME(SP3) * 1000);

IF NOT fbPowerCalcTimer.Q THEN
	fbPowerCalcTimer(IN := TRUE);
ELSE
	ulDeltaEnergy := ulInternalStorageValue - ulInternalStorageValueOld;	//Beräkna delta under samplingen

	IF (ulDeltaEnergy = 0) AND (rPower <> 0) AND (SP4 <> 0) THEN			//Om inget delta under samplingen och remanens är inställd, vänta ut remanenstimern innan värdet blir 0
		fbRemTimer(IN := TRUE, PT := UDINT_TO_TIME(SP4) * 1000);
		
		IF fbRemTimer.Q THEN
			rPower := 0;
		END_IF
	ELSE
		rPower := ((ulDeltaEnergy * 3600) / SP3) * SP2;  						//Beräkna effekt per timme (Wh, kWh, MWh etc)
		fbRemTimer(IN := FALSE);
	END_IF;

	ulInternalStorageValueOld := ulInternalStorageValue;  				//Uppdatera senaste värde
	fbPowerCalcTimer(IN := FALSE);
END_IF;

END_FUNCTION_BLOCK

// oaksLibrary/Mätare/fbPulseMeterkWh
FUNCTION_BLOCK fbPulseMeterkWh
VAR_INPUT
	{attribute 'OPC.UA.DA' := '1'}
	SP1 AT %M* : REAL; //Inställd mätarställning~wp:[unit]kWh[format]0.0[trendoptions]i:300
END_VAR
VAR 
	{attribute 'OPC.UA.DA' := '1'}
	PV4 AT %I* : BOOL; //Pulsingång~wp:
END_VAR
VAR_OUTPUT
	{attribute 'OPC.UA.DA' := '1'}
	PV AT %M*  : REAL; //Aktuell mätarställning~wp:[unit]kWh[format]0.0[trendoptions]i:300
	{attribute 'OPC.UA.DA' := '1'}
	PV5 AT %M* : INT; //Klockslag vid senaste puls (12:01 visas som 1201)~wp:
END_VAR
VAR
	stTime		: tc2_ba.TIMESTRUCT;
	nActualDayCase	: INT;
	nActualHour 	: INT;
	nActualMinute 	: INT;
	
	FB_BA_GetTime01 : tc2_ba.FB_BA_GetTime; 
	FB_BA_ExtTiSt01 : tc2_ba.FB_BA_ExtTiSt;		

	rTempVar : REAL;
	fbCounterTrig : r_trig;
	FbDoubleControlledVariableReal1 : FbDoubleControlledVariableReal;
END_VAR
VAR PERSISTENT 
	rInternalStorageValue : REAL; // Internt värde
END_VAR
VAR_INPUT PERSISTENT
	{attribute 'OPC.UA.DA' := '1'}
	SP2 AT %M* : REAL := 0.001; //Uppräkning per puls (exempelvis 0.001kWh per puls)~wp:[unit]kWh[format]0.000000
END_VAR

	FB_BA_GetTime01(bEn :=TRUE);	
	stTime := FB_BA_GetTime01.stSysTi;

	nActualDayCase :=WORD_TO_INT (stTime.wDayOfWeek);
	nActualHour :=WORD_TO_INT (stTime.wHour)*100;
	nActualMinute :=WORD_TO_INT (stTime.wMinute);

fbCounterTrig(CLK:=PV4 , Q=> );

IF fbCounterTrig.Q THEN 
	rTempVar := rInternalStorageValue + SP2;
	rInternalStorageValue := rTempVar;
	PV5 := nActualHour+nActualMinute;
END_IF


FbDoubleControlledVariableReal1(rVariableInPLC:=SP1 , rVariableInModbusUnit:= rInternalStorageValue);

PV := rInternalStorageValue;

END_FUNCTION_BLOCK

// oaksLibrary/Mätare/fbPulseMeterM3
FUNCTION_BLOCK fbPulseMeterM3
VAR_INPUT
	{attribute 'OPC.UA.DA' := '1'}
	SP1 AT %M* : REAL; //Inställd mätarställning~wp:[unit]m3[format]0.000000
END_VAR
VAR 
	{attribute 'OPC.UA.DA' := '1'}
	PV4 AT %I* : BOOL; //Pulsingång~wp:
END_VAR
VAR_OUTPUT
	{attribute 'OPC.UA.DA' := '1'}
	PV AT %M*  : REAL; //Aktuell mätarställning~wp:[unit]m3[format]0.00[trendoptions]i:300
	{attribute 'OPC.UA.DA' := '1'}
	PV5 AT %M* : INT; //Klockslag vid senaste puls (12:01 visas som 1201)~wp:
END_VAR
VAR
	stTime		: tc2_ba.TIMESTRUCT;
	nActualDayCase	: INT;
	nActualHour 	: INT;
	nActualMinute 	: INT;
	
	FB_BA_GetTime01 : tc2_ba.FB_BA_GetTime; 
	FB_BA_ExtTiSt01 : tc2_ba.FB_BA_ExtTiSt;		

	rTempVar : REAL;
	fbCounterTrig : r_trig;
	FbDoubleControlledVariableReal1 : FbDoubleControlledVariableReal;
END_VAR
VAR PERSISTENT 
	rInternalStorageValue : REAL; // Internt värde
END_VAR
VAR_INPUT PERSISTENT
	{attribute 'OPC.UA.DA' := '1'}
	SP2 AT %M* : REAL := 0.001; //Uppräkning per puls (exempelvis 0.001m3 per puls)~wp:[unit]m3[format]0.000000
END_VAR

	FB_BA_GetTime01(bEn :=TRUE);	
	stTime := FB_BA_GetTime01.stSysTi;

	nActualDayCase :=WORD_TO_INT (stTime.wDayOfWeek);
	nActualHour :=WORD_TO_INT (stTime.wHour)*100;
	nActualMinute :=WORD_TO_INT (stTime.wMinute);

fbCounterTrig(CLK:=PV4 , Q=> );

IF fbCounterTrig.Q THEN 
	rTempVar := rInternalStorageValue + SP2;
	rInternalStorageValue := rTempVar;
	PV5 := nActualHour+nActualMinute;
END_IF


FbDoubleControlledVariableReal1(rVariableInPLC:=SP1 , rVariableInModbusUnit:= rInternalStorageValue);

PV := rInternalStorageValue;

END_FUNCTION_BLOCK

// oaksLibrary/Mätare/fbPulseMeterMWh
FUNCTION_BLOCK fbPulseMeterMWh
VAR_INPUT
	{attribute 'OPC.UA.DA' := '1'}
	SP1 AT %M* : REAL; //Inställd mätarställning~wp:[unit]MWh[format]0.000000
END_VAR
VAR 
	{attribute 'OPC.UA.DA' := '1'}
	PV4 AT %I* : BOOL; //Pulsingång~wp:
END_VAR
VAR_OUTPUT
	{attribute 'OPC.UA.DA' := '1'}
	PV AT %M*  : REAL; //Aktuell mätarställning~wp:[unit]MWh[format]0.00[trendoptions]i:300
	{attribute 'OPC.UA.DA' := '1'}
	PV5 AT %M* : INT; //Klockslag vid senaste puls (12:01 visas som 1201)~wp:
END_VAR
VAR
	stTime		: tc2_ba.TIMESTRUCT;
	nActualDayCase	: INT;
	nActualHour 	: INT;
	nActualMinute 	: INT;
	
	FB_BA_GetTime01 : tc2_ba.FB_BA_GetTime; 
	FB_BA_ExtTiSt01 : tc2_ba.FB_BA_ExtTiSt;		

	rTempVar : REAL;
	fbCounterTrig : r_trig;
	FbDoubleControlledVariableReal1 : FbDoubleControlledVariableReal;
END_VAR
VAR PERSISTENT 
	rInternalStorageValue : REAL; // Internt värde
END_VAR
VAR_INPUT PERSISTENT
	{attribute 'OPC.UA.DA' := '1'}
	SP2 AT %M* : REAL := 0.001; //Uppräkning per puls (exempelvis 0.001MWh per puls)~wp:[unit]MWh[format]0.000000
END_VAR

	FB_BA_GetTime01(bEn :=TRUE);	
	stTime := FB_BA_GetTime01.stSysTi;

	nActualDayCase :=WORD_TO_INT (stTime.wDayOfWeek);
	nActualHour :=WORD_TO_INT (stTime.wHour)*100;
	nActualMinute :=WORD_TO_INT (stTime.wMinute);

fbCounterTrig(CLK:=PV4 , Q=> );

IF fbCounterTrig.Q THEN 
	rTempVar := rInternalStorageValue + SP2;
	rInternalStorageValue := rTempVar;
	PV5 := nActualHour+nActualMinute;
END_IF


FbDoubleControlledVariableReal1(rVariableInPLC:=SP1 , rVariableInModbusUnit:= rInternalStorageValue);

PV := rInternalStorageValue;

END_FUNCTION_BLOCK

// oaksLibrary/Mätare/fbPulseMeterV_Q
//Pulsräknare för beräkning av volym samt momentant flöde med tidsfaktor och remanens.
//Blocket är enhetsagnostiskt. För att få önskad enhet kan du antingen ställa in faktorn för uppräkning så att det motsvarar den enhet du önskar:
//	- t ex om mätaren pulsar liter och du vill ha m3 ställer du pulsfaktor på 0.001
//Eller så kan du ställa pulsfaktorn på 1, blocket kommer då räkna liter, sen kan du dela utvariabeln rVolume med 1000 för att få önskad enhet.
//Vill du ha olika storhet på räknaren och momentana värdet får du använda båda metoderna:
// - t ex för att få volym i m3 och flöde i l/h och mätaren pulsar liter, så ställer du pulsfaktorn till 0.001. Sen gångrar du rFlow med 1000.
//Samplingstid på 60s funkar i de flesta fall. Remanens används för att undvika att det momentana värdet faller till 0 direkt om det går längre tid än samplingstiden mellan pulser.
//Manuell omställning av mätaren kan göras på SP1. Ställ värdet till minst 1 (0 kommer ej att uppdatera räknaren)
//OAKS, 23-11-01

FUNCTION_BLOCK fbPulseMeterV_Q
VAR_INPUT
	bPulse AT %I* : BOOL; //Pulsingång
	{attribute 'OPC.UA.DA' := '1'}
	SP1 AT %M* : LREAL := 1; //Nytt värde mätarställning (obs lägst 1)~wp:[format]0.000
END_VAR

VAR_OUTPUT
	{attribute 'OPC.UA.DA' := '1'}
	PV5 AT %M* : INT; //Klockslag vid senaste puls volym~wp:

	lrVolume	: REAL; 	//Volym
	rFlow  		: REAL; 	//Beräknat flöde

	{attribute 'OPC.UA.DA' := '1'}
	FAULT  AT %M* : BOOL; //Samplingstid/pulsfaktor får ej vara 0~wp:
END_VAR
VAR
	stTime		: tc2_ba.TIMESTRUCT;
	nActualDayCase	: INT;
	nActualHour 	: INT;
	nActualMinute 	: INT;
	
	FB_BA_GetTime01 : tc2_ba.FB_BA_GetTime; 		

	fbCounterTrig : r_trig;
	
	ulInternalStorageValueOld : ULINT;
	
	fbFlowCalcTimer : TON;
	ulDelta : ULINT;
	fbRemTimer : TON;
	
	fbEdge : fbEdge;
END_VAR
VAR PERSISTENT 
	ulInternalStorageValue : ULINT; // Internt värde
END_VAR
VAR_INPUT PERSISTENT
	{attribute 'OPC.UA.DA' := '1'}
	SP2 AT %M* : REAL := 1; //Pulsfaktor (t ex 0.001 för m3 om mätarens pulsenhet är liter)~wp:
	{attribute 'OPC.UA.DA' := '1'}
	SP3 AT %M* : UDINT := 60; //Samplingstid för flödesberäkning~wp:[unit]s[format]0
	{attribute 'OPC.UA.DA' := '1'}
	SP4 AT %M* : UDINT := 0; //Remanens för flödesberäkning~wp:[unit]s[format]0
END_VAR

IF SP3 = 0 THEN
	SP3 := 1;
END_IF

IF SP2 = 0 THEN
	SP2 := 1;
END_IF

FAULT := (SP3 = 0) OR (SP2 = 0);

FB_BA_GetTime01(bEn :=TRUE);	
stTime := FB_BA_GetTime01.stSysTi;

nActualDayCase :=WORD_TO_INT (stTime.wDayOfWeek);
nActualHour :=WORD_TO_INT (stTime.wHour)*100;
nActualMinute :=WORD_TO_INT (stTime.wMinute);

//Beräkning volym
fbCounterTrig(CLK:=bPulse , Q=> );

IF fbCounterTrig.Q THEN 
	ulInternalStorageValue := ulInternalStorageValue + 1;
	PV5 := nActualHour+nActualMinute;
END_IF

lrVolume := ULINT_TO_LREAL(ulInternalStorageValue) * SP2;

fbEdge(anyInput := SP1);

IF fbEdge.bEdgeF AND SP1 <> 0 THEN
	ulInternalStorageValue := LREAL_TO_ULINT(SP1 / SP2);
	SP1 := 0;
 	ulInternalStorageValueOld := ulInternalStorageValue;
END_IF

//Beräkning flöde
fbFlowCalcTimer(PT := UDINT_TO_TIME(SP3) * 1000);

IF NOT fbFlowCalcTimer.Q THEN
	fbFlowCalcTimer(IN := TRUE);
ELSE
	ulDelta := ulInternalStorageValue - ulInternalStorageValueOld;	//Beräkna delta under samplingen

	IF (ulDelta = 0) AND (rFlow <> 0) AND (SP4 <> 0) THEN			//Om inget delta under samplingen och remanens är inställd, vänta ut remanenstimern innan värdet blir 0
		fbRemTimer(IN := TRUE, PT := UDINT_TO_TIME(SP4) * 1000);
		
		IF fbRemTimer.Q THEN
			rFlow := 0;
		END_IF
	ELSE
		rFlow := ((ulDelta * 3600) / SP3) * SP2;  						//Beräkna flöde per timme (m3/h, l/h etc)
		fbRemTimer(IN := FALSE);
	END_IF;

	ulInternalStorageValueOld := ulInternalStorageValue;  				//Uppdatera senaste värde
	fbFlowCalcTimer(IN := FALSE);
END_IF;

END_FUNCTION_BLOCK

// oaksLibrary/Mätare/fbPulseMeterV_Q_E_P
//Pulsräknare för beräkning av energi och volym samt momentan effekt och flöde med tidsfaktor och remanens.
//Blocket är enhetsagnostiskt. För att få önskad enhet kan du antingen ställa in faktorn för uppräkning så att det motsvarar den enhet du önskar:
//	- t ex om mätaren pulsar Wh och du vill ha kW ställer du pulsfaktor på 0.001
//Eller så kan du ställa pulsfaktorn på 1, blocket kommer då räkna Wh, sen kan du dela utvariabeln rEnergy med 1000 för att få önskad enhet.
//Vill du ha olika storhet på räknaren (t ex energi) och momentana värdet (t ex effekt) får du använda båda metoderna:
// - t ex för att få energi i MWh och effekt i kWh och mätaren pulsar kWh, så ställer du pulsfaktorn till 0.001. Sen gångrar du rPower med 1000.
//Samplingstid på 60s funkar i de flesta fall. Remanens används för att undvika att det momentana värdet faller till 0 direkt om det går längre tid än samplingstiden mellan pulser.
//Manuell omställning av mätaren kan göras på SP1 / SP5. Ställ värdet till minst 1 (0 kommer ej att uppdatera räknaren)
//OAKS, 23-11-01

FUNCTION_BLOCK fbPulseMeterV_Q_E_P
VAR_INPUT
	bVolPulse AT %I* : BOOL; //Pulsingång volym
	bEnPulse AT %I* : BOOL; //Pulsingång energi
	{attribute 'OPC.UA.DA' := '1'}
	SP1 AT %M* : LREAL := 1; //Nytt värde mätarställning volym (obs lägst 1)~wp:[format]0.000
	{attribute 'OPC.UA.DA' := '1'}
	SP5 AT %M* : LREAL := 1; //Nytt värde mätarställning energi (obs lägst 1)~wp:[format]0.000
END_VAR

VAR_OUTPUT
	{attribute 'OPC.UA.DA' := '1'}
	PV5 AT %M* : INT; //Klockslag vid senaste puls volym~wp:
	{attribute 'OPC.UA.DA' := '1'}
	PV7 AT %M* : INT; //Klockslag vid senaste puls energi~wp:	

	lrVolume	: REAL; 	//Volym
	rFlow  		: REAL; 	//Beräknat flöde
	lrEnergy	: REAL; 	//Energi
	rPower  	: REAL; 	//Beräknad effekt

	{attribute 'OPC.UA.DA' := '1'}
	FAULT  AT %M* : BOOL; //Samplingstid/pulsfaktor får ej vara 0~wp:
END_VAR
VAR
	stTime		: tc2_ba.TIMESTRUCT;
	nActualDayCase	: INT;
	nActualHour 	: INT;
	nActualMinute 	: INT;
	
	FB_BA_GetTime01 : tc2_ba.FB_BA_GetTime; 		

	fbCounterTrigVol : r_trig;
	
	fbCounterTrigEn : r_trig;
	
	ulInternalStorageValueVolOld : ULINT;
	
	ulInternalStorageValueEnOld : ULINT;
	
	fbFlowCalcTimer : TON;
	fbPowerCalcTimer : TON;
	ulDeltaVol : ULINT;
	ulDeltaEnergy : ULINT;
	fbRemTimerFlw : TON;
	fbRemTimerPwr : TON;
	
	fbEdgeVol : fbEdge;
	fbEdgeEn : fbEdge;
	
	iTest : INT;
END_VAR
VAR PERSISTENT 
	ulInternalStorageValueVol : ULINT; // Internt värde
	ulInternalStorageValueEn : ULINT; // Internt värde
END_VAR
VAR_INPUT PERSISTENT
	{attribute 'OPC.UA.DA' := '1'}
	SP2 AT %M* : REAL := 1; //Pulsfaktor volym (t ex 0.001 för m3 om mätarens pulsenhet är liter)~wp:
	{attribute 'OPC.UA.DA' := '1'}
	SP3 AT %M* : UDINT := 60; //Samplingstid för flödesberäkning~wp:[unit]s[format]0
	{attribute 'OPC.UA.DA' := '1'}
	SP4 AT %M* : UDINT := 0; //Remanens för flödesberäkning~wp:[unit]s[format]0
	{attribute 'OPC.UA.DA' := '1'}
	SP6 AT %M* : REAL := 1; //Pulsfaktor energi (t ex 0.001 för kWh om mätarens pulsenhet är Wh)~wp:
	{attribute 'OPC.UA.DA' := '1'}
	SP7 AT %M* : UDINT := 60; //Samplingstid för effektberäkning~wp:[unit]s[format]0
	{attribute 'OPC.UA.DA' := '1'}
	SP8 AT %M* : UDINT := 0; //Remanens för effektberäkning~wp:[unit]s[format]0
END_VAR

IF SP3 = 0 THEN
	SP3 := 1;
END_IF

IF SP2 = 0 THEN
	SP2 := 1;
END_IF

IF SP7 = 0 THEN
	SP7 := 1;
END_IF

IF SP6 = 0 THEN
	SP6 := 1;
END_IF

FAULT := (SP3 = 0) OR (SP7 = 0) OR (SP2 = 0) OR (SP6 = 0);

FB_BA_GetTime01(bEn :=TRUE);	
stTime := FB_BA_GetTime01.stSysTi;

nActualDayCase :=WORD_TO_INT (stTime.wDayOfWeek);
nActualHour :=WORD_TO_INT (stTime.wHour)*100;
nActualMinute :=WORD_TO_INT (stTime.wMinute);

//Beräkning volym
fbCounterTrigVol(CLK:=bVolPulse , Q=> );

IF fbCounterTrigVol.Q THEN 
	ulInternalStorageValueVol := ulInternalStorageValueVol + 1;
	PV5 := nActualHour+nActualMinute;
END_IF

lrVolume := ULINT_TO_LREAL(ulInternalStorageValueVol) * SP2;

fbEdgeVol(anyInput := SP1);

IF fbEdgeVol.bEdgeF AND SP1 <> 0 THEN
	ulInternalStorageValueVol := LREAL_TO_ULINT(SP1 / SP2);
	SP1 := 0;
 	ulInternalStorageValueVolOld := ulInternalStorageValueVol;
	iTest := iTest +1;
END_IF

//Beräkning flöde
fbFlowCalcTimer(PT := UDINT_TO_TIME(SP3) * 1000);

IF NOT fbFlowCalcTimer.Q THEN
	fbFlowCalcTimer(IN := TRUE);
ELSE
	ulDeltaVol := ulInternalStorageValueVol - ulInternalStorageValueVolOld;	//Beräkna delta under samplingen

	IF (ulDeltaVol = 0) AND (rFlow <> 0) AND (SP4 <> 0) THEN			//Om inget delta under samplingen och remanens är inställd, vänta ut remanenstimern innan värdet blir 0
		fbRemTimerFlw(IN := TRUE, PT := UDINT_TO_TIME(SP4) * 1000);
		
		IF fbRemTimerFlw.Q THEN
			rFlow := 0;
		END_IF
	ELSE
		rFlow := ((ulDeltaVol * 3600) / SP3) * SP2;  						//Beräkna flöde per timme (m3/h, l/h etc)
		fbRemTimerFlw(IN := FALSE);
	END_IF;

	ulInternalStorageValueVolOld := ulInternalStorageValueVol;  				//Uppdatera senaste värde
	fbFlowCalcTimer(IN := FALSE);
END_IF;



//Beräkning energi
fbCounterTrigEn(CLK:=bEnPulse , Q=> );

IF fbCounterTrigEn.Q THEN 
	ulInternalStorageValueEn := ulInternalStorageValueEn + 1;
	PV7 := nActualHour+nActualMinute;
END_IF

lrEnergy := ULINT_TO_LREAL(ulInternalStorageValueEn) * SP6;

fbEdgeEn(anyInput := SP5);

IF fbEdgeEn.bEdgeF AND SP5 <> 0 THEN
	ulInternalStorageValueEn := LREAL_TO_ULINT(SP5 / SP6);
	SP5 := 0;
 	ulInternalStorageValueEnOld := ulInternalStorageValueEn;
END_IF

//Beräkning effekt
fbPowerCalcTimer(PT := UDINT_TO_TIME(SP7) * 1000);

IF NOT fbPowerCalcTimer.Q THEN
	fbPowerCalcTimer(IN := TRUE);
ELSE
	ulDeltaEnergy := ulInternalStorageValueEn - ulInternalStorageValueEnOld;	//Beräkna delta under samplingen

	IF (ulDeltaEnergy = 0) AND (rPower <> 0) AND (SP8 <> 0) THEN			//Om inget delta under samplingen och remanens är inställd, vänta ut remanenstimern innan värdet blir 0
		fbRemTimerPwr(IN := TRUE, PT := UDINT_TO_TIME(SP8) * 1000);
		
		IF fbRemTimerPwr.Q THEN
			rPower := 0;
		END_IF
	ELSE
		rPower := ((ulDeltaEnergy * 3600) / SP7) * SP6;  						//Beräkna effekt per timme (Wh, kWh, MWh etc)
		fbRemTimerPwr(IN := FALSE);
	END_IF;

	ulInternalStorageValueEnOld := ulInternalStorageValueEn;  				//Uppdatera senaste värde
	fbPowerCalcTimer(IN := FALSE);
END_IF;

END_FUNCTION_BLOCK

// oaksLibrary/Poseidon/fbMotorRadMeanTempPoseidon
(*
Pumpstoppsfunktion VS pumpar.
För funktionen används maxvärde av två utetemperaturer.
Dels medeltemperatur över 72 timmar och aktuell utetemperatur.
Detta maxvärde stoppar och startar pumpen enligt i DUC inställbara värden.
En säkerhetsfunktion skall finnas som startar pumpen direkt vid lägre aktuell utetemperatur.
Efter start från säkerhetsfunktionen skall pumpen fortsatt vara i drift tills normal ute-stopptemperatur uppnåtts. 
Samtliga börvärde skall vara ändringsbara från ÖS.

*)
FUNCTION_BLOCK fbMotorRadMeanTempPoseidon EXTENDS fbMotor
VAR_INPUT
	rOutdoorTemp : ANY; // Utetemperatur används för start/stopp Knyter man inget här används oaksGVL.rOutdoortemp
	rOutdoorTempMean : ANY; // Knyt utemedeltemperatur
END_VAR
VAR_OUTPUT
	{attribute 'OPC.UA.DA' := '1'}
	PV4  AT %M*  : BOOL; //Startvillkor momentan utetemperatur under 5°C ~wp:[trendoptions]i:14400, t:1
	{attribute 'OPC.UA.DA' := '1'}
	PV5  AT %M*  : BOOL; //Startvillkor momentan utetemperatur under inställbart värde~wp:[trendoptions]i:14400, t:1
	{attribute 'OPC.UA.DA' := '1'}
	PV6  AT %M*  : BOOL; //Startvillkor medel utetemperatur under inställbart värde~wp:[trendoptions]i:14400, t:1
END_VAR
VAR
	rTempUsedMean : REAL; // Uteluftstemperatur medel
	rTempUsedMomentan : REAL; // Uteluftstemperatur
	fbPumpstoppTof : TOF;
	fbPumpstoppTon : TON;
END_VAR
VAR_INPUT PERSISTENT
	{attribute 'OPC.UA.DA' := '1'}
	SP2 AT %M* : INT := 15; //Stoppfördröjning~wp:[unit]min
	{attribute 'OPC.UA.DA' := '1'}
	SP1 AT %M* : REAL := 15;  //Stoppa pump om momentan eller medeltemperatur överstiger~wp:[unit]°C[format]0.0
	{attribute 'OPC.UA.DA' := '1'}
	SP3 AT %M* : INT := 180; //Startfördröjning~wp:[unit]min
END_VAR

	SUPER^();

	bStart := mStartPump();

(*
Pumpstoppsfunktion VS pumpar.
För funktionen används maxvärde av två utetemperaturer.
Dels medeltemperatur över 72 timmar och aktuell utetemperatur.
Detta maxvärde stoppar och startar pumpen enligt i DUC inställbara värden.
En säkerhetsfunktion skall finnas som startar pumpen direkt vid lägre aktuell utetemperatur.
Efter start från säkerhetsfunktionen skall pumpen fortsatt vara i drift tills normal ute-stopptemperatur uppnåtts. 
Samtliga börvärde skall vara ändringsbara från ÖS.

*)
// EJ KLART
METHOD PRIVATE mStartPump : BOOL
VAR_INPUT
END_VAR
VAR

	bTemperaturStart : BOOL;
	bOffDelayActive :  BOOL; //Aktiv stoppfördröjning av pump
	bOnDelayActive :  BOOL; //Aktiv startfördröjning av pump
END_VAR
//Temp select
rTempUsedMomentan := F_GetTempToUse(rOutdoorTemp);
rTempUsedMean := F_GetTempToUseMeanTemp(rOutdoorTempMean);
IF  rTempUsedMomentan < 5 THEN
	PV4 := TRUE;
ELSIF rTempUsedMomentan > SP1 THEN
	PV4 := FALSE;
END_IF
PV5 := rTempUsedMomentan < SP1;
PV6 := rTempUsedMean < SP1;
IF PV4 THEN //En Säkerhetsfunktion skall finnas som startar pumpen direkt vid lägre aktuell utetemperatur. Efter start från säkerhetsfunktionen skall pumpen fortsatt vara i drift tills normal ute-stopptemperatur uppnåtts. 
	bTemperaturStart := TRUE;
ELSIF PV5 AND PV6 THEN
	bTemperaturStart := TRUE;
ELSE
	bTemperaturStart := FALSE;
END_IF
fbPumpstoppTof(IN:=bTemperaturStart , PT:=fRealToMinute(SP2) , Q=> bOffDelayActive, ET=> );
fbPumpstoppTon(IN:=bTemperaturStart , PT:=fRealToMinute(SP3) , Q=> bOnDelayActive, ET=> );

//Starta pump
mStartPump := bOffDelayActive OR bOnDelayActive;
END_METHOD

END_FUNCTION_BLOCK

// oaksLibrary/Poseidon/fbPowerLimiterPoseidon
//Oaks AB
//2021-01-07
//Funktionsblock för effektbegräsning av temperatur för tex. VS/KB.
// Då utekompenserad effektbegränsning är aktiverad begränsas effekt till inställt värde genom att maxbegränsa värme/kylventilens öppningsgrad.
// Ärvärdets samplingstid är inställbart i Webport. Då effektbegränsning varit inkopplad i inställbar tid utgår larm. Blockering av effektbegränsning sker då lägsta rumstemperatur underskrider inställt värde.
FUNCTION_BLOCK fbPowerLimiterPoseidon
VAR_INPUT
	//Effektbegränsing
	rInstantaneousPower : REAL; //Momentaneffekt (kW)
	rOutdoorTemperature : REAL; // Utetemp
	rRoomTempLowest : REAL;
END_VAR

VAR_OUTPUT
	{attribute 'OPC.UA.DA' := '1'}
	CSP AT %M* : REAL; //Aktuell max-effekt~wp:[unit]kW[format]0.0
	//Effektbegränsning
	{attribute 'OPC.UA.DA' := '1'}
	PV AT %M* : REAL :=0; //Uträknat ärvärde effektbegränsning~wp:[unit]kW[format]0.0
	{attribute 'OPC.UA.DA' := '1'}
	PV4 AT %M* : REAL :=100; //Max utsignal värmeventil~wp:[unit]%[format]0
	{attribute 'OPC.UA.DA' := '1'}
	PV8 AT %M* : BOOL; //Driftvillkor rumstemperatur~wp:
	{attribute 'OPC.UA.DA' := '1'}
	AL AT %M* : BOOL; //Effektbegränsning lång aktiveringstid~wp:[alarmoptions]p:2
	{attribute 'OPC.UA.DA' := '1'}
	V AT %M* : BOOL; //Effektbegränsning aktiv~wp:[trendoptions]i:14400, t:1
	{attribute 'OPC.UA.DA' := '1'}
	PV5 AT %M* : BOOL; //Börvärdesförskjutning aktiverad~wp:
	
END_VAR

VAR
	fbTonRoomTemp : TON;	

	FB_BA_TiAvrg01 : tc2_ba.FB_BA_TiAvrg;
	
	iMedelvardeSekunder : UDINT;
	rkWhMax : REAL;
	rLimitOffset : REAL; //Förskjutning från effektbegränsning
	rProcentOffMax : REAL; 
	
	fbAlarmLimit: fbAlarm;
	fbController01: fbController;
	{attribute 'hide'}
	fbPushButtonBorvardesforskjutning : fbPushButton; // använder tryckknappsblock för att göra börvärdesförskjutning på inställd tid. lagt den som hide för att den inte ska dyka upp i webport eller io.
	fbResetTonM : TON; // Används för att återställa M-tagg
END_VAR

VAR_INPUT PERSISTENT
	{attribute 'OPC.UA.DA' := '1'}
	SP1 AT %M* :REAL:=19.5; //Tillåt effektbegränsning om lägsta rumstemperatur överstiger~wp:[unit]°C[format]0.0
	{attribute 'OPC.UA.DA' := '1'}
	SP3 AT %M* : UDINT := 40; //Tid för medelvärdesberäkning effekt för effektbegränsning (1-256)~wp:[unit]sekunder[format]0
	{attribute 'OPC.UA.DA' := '1'}
	SP4 AT %M* : INT := 24; //Aktiveringstid börvärdesförskjutning~wp:[unit]h[format]0
	{attribute 'OPC.UA.DA' := '1'}
	SP5 AT %M* : REAL := 3; //Börvärdesförskjutning (då börvärdesförskjutning aktiv)~wp:[unit]KW[format]0
	
	{attribute 'OPC.UA.DA' := '1'}
	P AT %M* : REAL := 0.3;  //Förstärkning~wp:[format]0.00
	{attribute 'OPC.UA.DA' := '1'}
	I AT %M* : UDINT := 300; //I-tid~wp:
	{attribute 'OPC.UA.DA' := '1'}
	DZ AT %M* : REAL := 0.1; //Dödzon~wp:[format]0.00

	{attribute 'OPC.UA.DA' := '1'}
	Y1 AT %M* : REAL:=500; //Max effekt/Utetemp~wp:[unit]kW[format]0.0
	{attribute 'OPC.UA.DA' := '1'}
	Y2 AT %M* :	REAL:=500; //Max effekt/Utetemp~wp:[unit]kW[format]0.0
	{attribute 'OPC.UA.DA' := '1'}
	Y3 AT %M* :	REAL:=500; //Max effekt/Utetemp~wp:[unit]kW[format]0.0
	{attribute 'OPC.UA.DA' := '1'}
	Y4 AT %M* :	REAL:=500; //Max effekt/Utetemp~wp:[unit]kW[format]0.0
	{attribute 'OPC.UA.DA' := '1'}
	Y5 AT %M* :	REAL:=500; //Max effekt/Utetemp~wp:[unit]kW[format]0.0
	{attribute 'OPC.UA.DA' := '1'}
	Y6 AT %M* :	REAL:=500; //Max effekt/Utetemp~wp:[unit]kW[format]0.0
	{attribute 'OPC.UA.DA' := '1'}
	X1 AT %M* :	REAL:=-30; //Utetemperatur~wp:[unit]°C[format]0.0
	{attribute 'OPC.UA.DA' := '1'}
	X2 AT %M* :	REAL:=-20; //Utetemperatur~wp:[unit]°C[format]0.0
	{attribute 'OPC.UA.DA' := '1'}
	X3 AT %M* :	REAL:=-10; //Utetemperatur~wp:[unit]°C[format]0.0
	{attribute 'OPC.UA.DA' := '1'}
	X4 AT %M* :	REAL:=0; //Utetemperatur~wp:[unit]°C[format]0.0
	{attribute 'OPC.UA.DA' := '1'}
	X5 AT %M* :	REAL:=10; //Utetemperatur~wp:[unit]°C[format]0.0
	{attribute 'OPC.UA.DA' := '1'}
	X6 AT %M* :	REAL:=20; //Utetemperatur~wp:[unit]°C[format]0.0


	M AT %M* : BOOL := FALSE; //Aktivering tidsinställd börvärdesförskjutning~wp:[trendoptions]i:14400, t:1
	
	//Effektstyrning
	{attribute 'OPC.UA.DA' := '1'}
	MO AT %M* : BOOL := FALSE; //Aktivering effektbegränsning~wp:[trendoptions]i:14400, t:1
	{attribute 'OPC.UA.DA' := '1'}
	AD AT %M* : REAL :=12; //Larmfördröjning lång inkopplingstid effektbegränsning~wp:[unit]timmar[format]0
	
END_VAR

	IF SP3 > 256 THEN // Medelvärdestid maxbegränsas till 256 sekunder.
		SP3 := 256;
	ELSIF SP3 < 1 THEN // Medelvärdestid minbegränsas till 2 sekunder.
		SP3 := 1;
	END_IF
	
	IF SP3 <= 256 AND SP3 > 0 THEN
		 iMedelvardeSekunder := SP3;
	END_IF;

	fbTonRoomTemp(IN:=rRoomTempLowest > SP1 , PT:=T#1M , Q=>PV8 , ET=> );

	
	
	//Tidsinställd börvärdesförskjutning vid aktivering
	IF M THEN
		fbResetTonM.IN := TRUE;
		IF fbResetTonM.Q THEN
			M := FALSE;
		END_IF
	ELSE
		fbResetTonM.IN := FALSE;
	END_IF
	fbResetTonM.PT := T#0.5S;
	fbResetTonM();
	
	fbPushButtonBorvardesforskjutning(SP1:=SP4*60,M:= M);
	PV5 := fbPushButtonBorvardesforskjutning.V;
	//Uträknat börvärde
	IF PV5 THEN
		CSP := fScale6p(rX:= rOutdoorTemperature, Y1:= Y1, Y2:= Y2, Y3:= Y3, Y4:= Y4, Y5:= Y5, Y6:= Y6, X1:= X1, X2:= X2, X3:= X3, X4:= X4, X5:= X5, X6:= X6) + SP5;
	ELSE
		CSP := fScale6p(rX:= rOutdoorTemperature, Y1:= Y1, Y2:= Y2, Y3:= Y3, Y4:= Y4, Y5:= Y5, Y6:= Y6, X1:= X1, X2:= X2, X3:= X3, X4:= X4, X5:= X5, X6:= X6);
	END_IF

	
	FB_BA_TiAvrg01(
	bEn:= TRUE, 
	bEnAvrg := TRUE,
	lrIn:=REAL_TO_LREAL(rInstantaneousPower), 
	udiIntval:=1, 
	udiNumOfElem:= iMedelvardeSekunder, 
	lrOut=> );
	
	PV := LREAL_TO_REAL(FB_BA_TiAvrg01.lrOut);
	fbController01(
	bEnable:= MO AND PV8, 
	rProcessValue:= PV, 
	rSetpoint:=CSP , 
	bActn:= FALSE, 
	rKp:= P, 
	rKi:= I, 
	rDz:= DZ, 
	rMin:= 0, 
	rMax:= 100, 
	rOutput=> );
	IF fbController01.bEnable THEN
		PV4 := fbController01.rOutput;
	ELSE
		PV4 := 100;
	END_IF

	//Indikering effektbegränsning aktiv
	IF fbController01.rOutput < 100 AND fbController01.bEnable THEN
		V := TRUE;
	ELSE 
		V := FALSE;
	END_IF
	
	//Larm lång inkopplingstid
	fbAlarmLimit(bInput:= V, tAlarmDelay:= fRealToHour(AD), bAutoReset:= TRUE, bAlarmOutput=> AL);

END_FUNCTION_BLOCK

// oaksLibrary/Regulatorer/fbController
// Pi-regulator. 
{attribute 'initialize_on_call'}
FUNCTION_BLOCK fbController
VAR_INPUT
	bEnable : BOOL; // Aktiverar reglering
	bPause : BOOL; // Pausa regulator
	rProcessValue : REAL; // Aktuellt Ärvärde 
	rSetpoint : REAL; // Aktuellt börvärde
	bActn : BOOL; // Gångriktning reglersekvens (kylsekvens = TRUE)
	rKp : REAL; // Kp
	rKi : UDINT; // Ki
	rDi : UDINT; // D-tid (Derivata)
	rFDi : UDINT; // Filter tid D (Derivata)
	rDz : REAL :=0.4; //Dödzon
	rMin : REAL := 0; // min reglersignal
	rMax : REAL := 100; // max reglersignal
	rSync : REAL := 0; 	// Synk-värde
	rOffVal : REAL := 0; //Utgång om ej bEnable
	bSync : BOOL;	// Synk-kommando
	{attribute 'pingroup' := 'DeviationAlarm'}
	{attribute 'initialize_on_call'}
	rDevLimit : REFERENCE TO REAL := 0;
	{attribute 'pingroup' := 'DeviationAlarm'}
	bBlockHighAlarm : BOOL; // Blockera högtemplarm
	{attribute 'pingroup' := 'DeviationAlarm'}
	bBlockLowAlarm : BOOL; // Blockera lågtemplarm
	{attribute 'pingroup' := 'DeviationAlarm'}
	tAlarmDelay : TIME := T#5S; // larmfördröjning
END_VAR
VAR_OUTPUT
	rOutput : REAL; // regulatorsignal
	{attribute 'pingroup' := 'DeviationAlarm'}
	bAlarmOutput : BOOL; //larmutgång
END_VAR
VAR
	fbReg01 : Tc3_BA_Common.FB_BA_PIDCtrl;
	fbDevAlarmPV: fbDevAlarm;
	rDevLimitInternal : REAL;
END_VAR


	fbDevAlarmPV(
	tAlarmDelay:=tAlarmDelay , 
	bAutoReset:=TRUE , 
	bAlarmOutput=>bAlarmOutput , 
	bEnable:=bEnable AND mDevAlarmCheck() ,
	rProcessValue:=rProcessValue , 
	rSetPoint:=rSetpoint , 
	rDevLimit:=rDevLimitInternal , 
	bBlockHighAlarm:=bBlockHighAlarm , 
	bBlockLowAlarm:=bBlockLowAlarm );

IF NOT bPause THEN
	fbReg01(
	bEn:=bEnable , 
	rW:=rSetpoint , 
	rX:=rProcessValue , 
	udiOpMode:= , 
	bActn:=bActn , 
	rKp:= rKp, 
	udiTn_ms:= rKi*1000, 
	udiTv_ms:=rDi*1000 , 
	udiTd_ms:=rFDi*1000 , 
	rYMax:= rMax, 
	rYMin:=rMin , 
	rNZ:=rDz , 
	udiCycCl:= , 
	bSync:=bSync, 
	rSync:=rSync,  
	rY=> , 
	rE=> , 
	bARW=> );
END_IF
	
IF bEnable THEN
	rOutput := fbReg01.rY;
ELSE
	rOutput := rOffVal;
END_IF

// Kolla ifall något är knutet på inputen rDevLimit. Är inget knutet där inaktiveras avvikelselarmet.
METHOD PRIVATE mDevAlarmCheck : BOOL // Valt börvärde
IF __ISVALIDREF(rDevLimit) THEN 
	mDevAlarmCheck := TRUE;
	rDevLimitInternal := rDevLimit;
ELSE
	mDevAlarmCheck := FALSE;
END_IF
END_METHOD

END_FUNCTION_BLOCK

